C03658=1182.878,246.002,-64.070,-177.311,7.140,148.552
C03659=1182.873,246.251,-64.098,-177.308,7.143,148.552
C03660=1182.869,246.499,-64.123,-177.305,7.145,148.551
C03661=1182.864,246.748,-64.150,-177.303,7.148,148.551
C03662=1182.860,246.996,-64.177,-177.300,7.150,148.551
C03663=1182.856,247.245,-64.204,-177.297,7.153,148.551
C03664=1182.851,247.493,-64.231,-177.295,7.155,148.551
C03665=1182.847,247.742,-64.257,-177.292,7.158,148.551
C03666=1182.842,247.990,-64.284,-177.290,7.160,148.551
C03667=1182.837,248.239,-64.311,-177.287,7.163,148.551
C03668=1182.834,248.487,-64.337,-177.285,7.165,148.550
C03669=1182.829,248.736,-64.364,-177.282,7.168,148.550
C03670=1182.824,248.984,-64.391,-177.279,7.170,148.550
C03671=1182.820,249.233,-64.418,-177.277,7.173,148.550
C03672=1182.815,249.481,-64.444,-177.274,7.175,148.550
C03673=1182.811,249.730,-64.471,-177.271,7.178,148.550
C03674=1182.806,249.978,-64.498,-177.269,7.181,148.550
C03675=1182.803,250.227,-64.525,-177.266,7.182,148.549
C03676=1182.798,250.476,-64.552,-177.263,7.185,148.549
C03677=1182.793,250.724,-64.579,-177.261,7.188,148.549
C03678=1182.789,250.973,-64.606,-177.258,7.190,148.549
C03679=1182.785,251.221,-64.633,-177.256,7.192,148.549
C03680=1182.780,251.469,-64.660,-177.253,7.195,148.549
C03681=1182.775,251.718,-64.687,-177.251,7.197,148.549
C03682=1182.771,251.966,-64.714,-177.248,7.200,148.548
C03683=1182.766,252.215,-64.741,-177.245,7.202,148.548
C03684=1182.763,252.464,-64.768,-177.243,7.205,148.548
C03685=1182.758,252.712,-64.795,-177.240,7.207,148.548
C03686=1182.754,252.961,-64.822,-177.237,7.210,148.548
C03687=1182.749,253.209,-64.850,-177.235,7.213,148.548
C03688=1182.745,253.457,-64.877,-177.232,7.215,148.548
C03689=1182.740,253.706,-64.904,-177.229,7.218,148.547
C03690=1182.737,253.955,-64.931,-177.227,7.220,148.547
C03691=1182.732,254.203,-64.958,-177.224,7.223,148.547
C03692=1182.727,254.452,-64.985,-177.222,7.225,148.547
C03693=1182.723,254.700,-65.012,-177.219,7.228,148.547
C03694=1182.718,254.948,-65.040,-177.216,7.231,148.547
C03695=1182.714,255.196,-65.067,-177.214,7.233,148.547
C03696=1182.710,255.446,-65.094,-177.211,7.236,148.546
C03697=1182.705,255.694,-65.121,-177.209,7.238,148.546
C03698=1182.700,255.943,-65.148,-177.206,7.241,148.546
C03699=1182.697,256.190,-65.176,-177.204,7.243,148.546
C03700=1182.692,256.439,-65.203,-177.201,7.245,148.546
C03701=1182.688,256.688,-65.230,-177.198,7.248,148.546
C03702=1182.684,256.936,-65.258,-177.196,7.251,148.546
C03703=1182.679,257.184,-65.285,-177.193,7.254,148.546
C03704=1182.674,257.433,-65.312,-177.190,7.255,148.545
C03705=1182.670,257.682,-65.339,-177.187,7.258,148.545
C03706=1182.666,257.930,-65.367,-177.185,7.261,148.545
C03707=1182.661,258.178,-65.394,-177.183,7.264,148.545
C03708=1182.657,258.427,-65.421,-177.179,7.266,148.545
C03709=1182.653,258.675,-65.449,-177.177,7.268,148.545
C03710=1182.648,258.924,-65.476,-177.174,7.271,148.545
C03711=1182.644,259.172,-65.504,-177.172,7.273,148.545
C03712=1182.639,259.420,-65.531,-177.170,7.276,148.545
C03713=1182.635,259.669,-65.559,-177.166,7.279,148.544
C03714=1182.631,259.917,-65.586,-177.164,7.281,148.544
C03715=1182.625,260.166,-65.614,-177.161,7.284,148.544
C03716=1182.622,260.415,-65.642,-177.159,7.287,148.544
C03717=1182.617,260.663,-65.669,-177.156,7.289,148.544
C03718=1182.613,260.911,-65.697,-177.153,7.292,148.544
C03719=1182.608,261.160,-65.725,-177.151,7.294,148.544
C03720=1182.604,261.408,-65.752,-177.148,7.297,148.544
C03721=1182.599,261.657,-65.779,-177.146,7.300,148.544
C03722=1182.596,261.905,-65.808,-177.143,7.302,148.543
C03723=1182.590,262.178,-65.838,-177.140,7.305,148.543
C03724=1182.586,262.451,-65.869,-177.138,7.308,148.543
C03725=1182.581,262.724,-65.899,-177.135,7.311,148.543
C03726=1182.577,262.997,-65.929,-177.132,7.314,148.543
C03727=1182.571,263.246,-65.957,-177.129,7.317,148.543
C03728=1182.567,263.493,-65.984,-177.127,7.319,148.543
C03729=1182.563,263.742,-66.012,-177.124,7.322,148.543
C03730=1182.558,263.991,-66.040,-177.121,7.324,148.542
C03731=1182.554,264.238,-66.067,-177.119,7.327,148.542
C03732=1182.550,264.487,-66.096,-177.116,7.329,148.542
C03733=1182.545,264.736,-66.123,-177.113,7.332,148.542
C03734=1182.541,264.984,-66.151,-177.111,7.335,148.542
C03735=1182.537,265.232,-66.179,-177.108,7.338,148.542
C03736=1182.532,265.481,-66.206,-177.106,7.339,148.542
C03737=1182.528,265.730,-66.235,-177.103,7.342,148.542
C03738=1182.523,265.977,-66.263,-177.100,7.345,148.542
C03739=1182.520,266.226,-66.291,-177.098,7.348,148.542
C03740=1182.514,266.475,-66.318,-177.095,7.351,148.542
C03741=1182.510,266.723,-66.346,-177.093,7.354,148.542
C03742=1182.506,266.971,-66.374,-177.090,7.356,148.541
C03743=1182.502,267.219,-66.402,-177.087,7.358,148.541
C03744=1182.497,267.469,-66.430,-177.085,7.361,148.541
C03745=1182.493,267.717,-66.458,-177.082,7.363,148.541
C03746=1182.489,267.965,-66.486,-177.080,7.366,148.541
C03747=1182.484,268.213,-66.514,-177.077,7.369,148.541
C03748=1182.479,268.461,-66.542,-177.075,7.372,148.541
C03749=1182.476,268.710,-66.570,-177.072,7.375,148.541
C03750=1182.471,268.958,-66.599,-177.069,7.378,148.541
C03751=1182.467,269.207,-66.626,-177.067,7.379,148.540
C03752=1182.462,269.455,-66.654,-177.064,7.382,148.540
C03753=1182.458,269.704,-66.683,-177.061,7.385,148.540
C03754=1182.453,269.952,-66.710,-177.059,7.388,148.540
C03755=1182.449,270.201,-66.739,-177.056,7.391,148.540
C03756=1182.445,270.449,-66.767,-177.054,7.394,148.540
C03757=1182.441,270.697,-66.795,-177.051,7.396,148.540
C03758=1182.436,270.945,-66.823,-177.049,7.399,148.540
C03759=1182.432,271.194,-66.852,-177.045,7.401,148.540
C03760=1182.427,271.442,-66.880,-177.043,7.403,148.540
C03761=1182.423,271.691,-66.908,-177.041,7.406,148.540
C03762=1182.418,271.939,-66.937,-177.038,7.409,148.540
C03763=1182.414,272.187,-66.965,-177.036,7.412,148.540
C03764=1182.409,272.436,-66.993,-177.033,7.415,148.540
C03765=1182.405,272.684,-67.021,-177.030,7.418,148.539
C03766=1182.402,272.932,-67.050,-177.028,7.420,148.539
C03767=1182.397,273.180,-67.078,-177.025,7.423,148.539
C03768=1182.393,273.429,-67.107,-177.023,7.426,148.539
C03769=1182.388,273.677,-67.135,-177.020,7.429,148.539
C03770=1182.384,273.926,-67.163,-177.017,7.431,148.539
C03771=1182.379,274.174,-67.191,-177.015,7.433,148.539
C03772=1182.375,274.423,-67.220,-177.012,7.436,148.539
C03773=1182.371,274.671,-67.248,-177.010,7.439,148.539
C03774=1182.366,274.919,-67.277,-177.007,7.442,148.539
C03775=1182.362,275.168,-67.306,-177.004,7.445,148.539
C03776=1182.357,275.416,-67.334,-177.002,7.447,148.539
C03777=1182.354,275.664,-67.362,-176.999,7.450,148.539
C03778=1182.349,275.913,-67.392,-176.997,7.453,148.539
C03779=1182.345,276.160,-67.419,-176.994,7.456,148.539
C03780=1182.341,276.409,-67.448,-176.992,7.458,148.538
C03781=1182.335,276.657,-67.476,-176.989,7.461,148.538
C03782=1182.332,276.905,-67.505,-176.986,7.464,148.538
C03783=1182.328,277.154,-67.534,-176.984,7.466,148.538
C03784=1182.322,277.403,-67.562,-176.981,7.469,148.538
C03785=1182.319,277.650,-67.591,-176.979,7.472,148.538
C03786=1182.315,277.899,-67.620,-176.976,7.475,148.538
C03787=1182.310,278.147,-67.648,-176.974,7.477,148.538
C03788=1182.306,278.395,-67.677,-176.971,7.480,148.538
C03789=1182.302,278.644,-67.706,-176.968,7.483,148.538
C03790=1182.297,278.892,-67.734,-176.965,7.486,148.538
C03791=1182.293,279.141,-67.763,-176.963,7.488,148.538
C03792=1182.288,279.389,-67.792,-176.960,7.491,148.538
C03793=1182.284,279.637,-67.820,-176.957,7.494,148.538
C03794=1182.280,279.886,-67.849,-176.955,7.496,148.538
C03795=1182.276,280.134,-67.879,-176.953,7.499,148.537
C03796=1182.271,280.382,-67.907,-176.950,7.502,148.537
C03797=1182.267,280.630,-67.936,-176.947,7.505,148.537
C03798=1182.263,280.879,-67.965,-176.945,7.507,148.537
C03799=1182.259,281.127,-67.994,-176.942,7.510,148.537
C03800=1182.253,281.375,-68.022,-176.939,7.513,148.537
C03801=1182.250,281.623,-68.051,-176.937,7.516,148.537
C03802=1182.246,281.872,-68.080,-176.935,7.518,148.537
C03803=1182.241,282.120,-68.109,-176.932,7.521,148.537
C03804=1182.236,282.369,-68.138,-176.929,7.524,148.537
C03805=1182.232,282.617,-68.167,-176.926,7.527,148.537
C03806=1182.229,282.865,-68.196,-176.924,7.529,148.537
C03807=1182.224,283.113,-68.224,-176.922,7.532,148.537
C03808=1182.219,283.361,-68.254,-176.919,7.535,148.537
C03809=1182.215,283.610,-68.283,-176.916,7.538,148.537
C03810=1182.211,283.858,-68.312,-176.914,7.541,148.537
C03811=1182.206,284.106,-68.341,-176.911,7.544,148.537
C03812=1182.201,284.355,-68.370,-176.908,7.547,148.537
C03813=1182.198,284.603,-68.399,-176.906,7.550,148.537
C03814=1182.194,284.851,-68.428,-176.904,7.552,148.537
C03815=1182.190,285.099,-68.458,-176.901,7.555,148.537
C03816=1182.185,285.348,-68.486,-176.899,7.558,148.537
C03817=1182.180,285.596,-68.516,-176.896,7.561,148.537
C03818=1182.176,285.844,-68.545,-176.893,7.564,148.537
C03819=1182.172,286.092,-68.574,-176.891,7.566,148.537
C03820=1182.168,286.341,-68.603,-176.888,7.569,148.537
C03821=1182.163,286.589,-68.632,-176.886,7.572,148.537
C03822=1182.159,286.837,-68.662,-176.883,7.575,148.536
C03823=1182.154,287.085,-68.691,-176.881,7.577,148.536
C03824=1182.150,287.334,-68.721,-176.878,7.580,148.536
C03825=1182.146,287.583,-68.749,-176.875,7.583,148.536
C03826=1182.142,287.831,-68.779,-176.872,7.586,148.536
C03827=1182.137,288.105,-68.811,-176.870,7.589,148.536
C03828=1182.132,288.380,-68.844,-176.867,7.592,148.536
C03829=1182.128,288.654,-68.876,-176.864,7.595,148.536
C03830=1182.123,288.929,-68.909,-176.862,7.598,148.536
C03831=1182.118,289.177,-68.938,-176.859,7.601,148.536
C03832=1182.114,289.426,-68.968,-176.856,7.604,148.536
C03833=1182.110,289.673,-68.997,-176.853,7.607,148.536
C03834=1182.105,289.921,-69.026,-176.851,7.610,148.536
C03835=1182.101,290.170,-69.056,-176.849,7.612,148.536
C03836=1182.097,290.418,-69.085,-176.846,7.615,148.536
C03837=1182.093,290.666,-69.115,-176.843,7.618,148.536
C03838=1182.089,290.914,-69.144,-176.841,7.622,148.536
C03839=1182.084,291.163,-69.173,-176.838,7.625,148.536
C03840=1182.080,291.411,-69.203,-176.836,7.627,148.536
C03841=1182.076,291.659,-69.232,-176.833,7.630,148.536
C03842=1182.072,291.908,-69.262,-176.830,7.633,148.536
C03843=1182.067,292.156,-69.292,-176.828,7.636,148.536
C03844=1182.063,292.404,-69.321,-176.825,7.639,148.536
C03845=1182.058,292.652,-69.350,-176.823,7.641,148.536
C03846=1182.054,292.900,-69.380,-176.820,7.644,148.536
C03847=1182.050,293.148,-69.409,-176.817,7.647,148.536
C03848=1182.046,293.396,-69.439,-176.815,7.650,148.536
C03849=1182.042,293.644,-69.469,-176.812,7.653,148.536
C03850=1182.037,293.893,-69.499,-176.810,7.655,148.536
C03851=1182.032,294.141,-69.528,-176.808,7.658,148.536
C03852=1182.028,294.390,-69.558,-176.805,7.661,148.536
C03853=1182.024,294.637,-69.588,-176.802,7.664,148.536
C03854=1182.020,294.885,-69.618,-176.799,7.667,148.536
C03855=1182.015,295.134,-69.648,-176.797,7.670,148.536
C03856=1182.011,295.382,-69.677,-176.795,7.673,148.536
C03857=1182.007,295.630,-69.707,-176.792,7.676,148.536
C03858=1182.003,295.878,-69.737,-176.790,7.679,148.536
C03859=1181.998,296.127,-69.767,-176.787,7.682,148.536
C03860=1181.994,296.375,-69.796,-176.784,7.685,148.536
C03861=1181.990,296.623,-69.826,-176.781,7.688,148.536
C03862=1181.986,296.871,-69.856,-176.779,7.690,148.536
C03863=1181.981,297.120,-69.886,-176.777,7.693,148.536
C03864=1181.978,297.368,-69.916,-176.774,7.696,148.536
C03865=1181.974,297.616,-69.946,-176.771,7.699,148.536
C03866=1181.969,297.864,-69.977,-176.769,7.702,148.536
C03867=1181.965,298.112,-70.006,-176.766,7.705,148.536
C03868=1181.961,298.361,-70.035,-176.764,7.707,148.536
C03869=1181.956,298.609,-70.066,-176.762,7.711,148.536
C03870=1181.952,298.857,-70.096,-176.759,7.714,148.536
C03871=1181.948,299.105,-70.126,-176.756,7.717,148.536
C03872=1181.943,299.353,-70.156,-176.753,7.720,148.536
C03873=1181.939,299.601,-70.186,-176.751,7.723,148.536
C03874=1181.935,299.849,-70.216,-176.749,7.725,148.536
C03875=1181.930,300.097,-70.246,-176.746,7.728,148.536
C03876=1181.926,300.345,-70.276,-176.744,7.731,148.536
C03877=1181.922,300.594,-70.307,-176.741,7.734,148.536
C03878=1181.918,300.842,-70.336,-176.738,7.737,148.536
C03879=1181.913,301.090,-70.367,-176.735,7.740,148.536
C03880=1181.909,301.338,-70.397,-176.734,7.743,148.536
C03881=1181.905,301.586,-70.427,-176.731,7.746,148.536
C03882=1181.900,301.835,-70.457,-176.728,7.749,148.536
C03883=1181.896,302.082,-70.487,-176.726,7.752,148.536
C03884=1181.892,302.330,-70.518,-176.723,7.755,148.536
C03885=1181.888,302.579,-70.548,-176.721,7.758,148.536
C03886=1181.884,302.827,-70.578,-176.718,7.761,148.536
C03887=1181.880,303.075,-70.608,-176.716,7.763,148.536
C03888=1181.875,303.323,-70.638,-176.713,7.766,148.536
C03889=1181.871,303.571,-70.669,-176.710,7.769,148.536
C03890=1181.866,303.819,-70.699,-176.708,7.772,148.536
C03891=1181.863,304.068,-70.729,-176.705,7.775,148.536
C03892=1181.858,304.316,-70.760,-176.703,7.778,148.536
C03893=1181.854,304.564,-70.790,-176.700,7.781,148.536
C03894=1181.849,304.812,-70.820,-176.698,7.785,148.536
C03895=1181.845,305.060,-70.851,-176.695,7.787,148.536
C03896=1181.841,305.308,-70.881,-176.693,7.790,148.536
C03897=1181.837,305.556,-70.912,-176.690,7.793,148.536
C03898=1181.833,305.804,-70.942,-176.688,7.796,148.536
C03899=1181.828,306.053,-70.972,-176.685,7.799,148.536
C03900=1181.823,306.301,-71.003,-176.682,7.802,148.536
C03901=1181.820,306.549,-71.034,-176.680,7.805,148.536
C03902=1181.816,306.797,-71.065,-176.677,7.808,148.537
C03903=1181.812,307.045,-71.095,-176.675,7.811,148.536
C03904=1181.807,307.292,-71.125,-176.672,7.814,148.536
C03905=1181.802,307.540,-71.156,-176.670,7.817,148.536
C03906=1181.799,307.789,-71.186,-176.667,7.820,148.537
C03907=1181.794,308.037,-71.217,-176.665,7.823,148.537
C03908=1181.790,308.285,-71.248,-176.662,7.826,148.537
C03909=1181.786,308.533,-71.278,-176.660,7.829,148.537
C03910=1181.782,308.782,-71.309,-176.657,7.832,148.537
C03911=1181.777,309.030,-71.340,-176.655,7.834,148.537
C03912=1181.773,309.277,-71.370,-176.652,7.837,148.537
C03913=1181.769,309.526,-71.401,-176.650,7.841,148.537
C03914=1181.765,309.774,-71.432,-176.647,7.844,148.537
C03915=1181.760,310.022,-71.462,-176.644,7.847,148.537
C03916=1181.757,310.270,-71.493,-176.642,7.850,148.537
C03917=1181.752,310.518,-71.524,-176.639,7.853,148.537
C03918=1181.748,310.766,-71.555,-176.637,7.856,148.537
C03919=1181.743,311.014,-71.585,-176.635,7.859,148.537
C03920=1181.740,311.262,-71.616,-176.632,7.861,148.537
C03921=1181.735,311.510,-71.647,-176.630,7.864,148.537
C03922=1181.731,311.758,-71.678,-176.627,7.868,148.537
C03923=1181.727,312.006,-71.709,-176.625,7.871,148.537
C03924=1181.722,312.254,-71.740,-176.622,7.874,148.537
C03925=1181.718,312.502,-71.770,-176.620,7.877,148.537
C03926=1181.714,312.751,-71.801,-176.617,7.880,148.537
C03927=1181.710,312.999,-71.832,-176.614,7.883,148.537
C03928=1181.706,313.247,-71.864,-176.612,7.886,148.538
C03929=1181.701,313.495,-71.895,-176.609,7.889,148.538
C03930=1181.697,313.743,-71.925,-176.607,7.892,148.538
C03931=1181.693,314.019,-71.960,-176.604,7.896,148.538
C03932=1181.688,314.296,-71.994,-176.602,7.899,148.538
C03933=1181.683,314.573,-72.029,-176.598,7.902,148.538
C03934=1181.678,314.849,-72.064,-176.596,7.905,148.538
C03935=1181.674,315.097,-72.095,-176.593,7.909,148.538
C03936=1181.670,315.345,-72.125,-176.591,7.912,148.538
C03937=1181.666,315.593,-72.157,-176.588,7.915,148.538
C03938=1181.661,315.841,-72.188,-176.586,7.918,148.538
C03939=1181.657,316.090,-72.219,-176.583,7.921,148.538
C03940=1181.653,316.337,-72.251,-176.581,7.924,148.538
C03941=1181.648,316.585,-72.281,-176.578,7.927,148.538
C03942=1181.644,316.834,-72.313,-176.576,7.930,148.538
C03943=1181.640,317.081,-72.344,-176.573,7.933,148.539
C03944=1181.637,317.330,-72.375,-176.571,7.936,148.539
C03945=1181.633,317.577,-72.406,-176.569,7.939,148.539
C03946=1181.629,317.826,-72.437,-176.566,7.942,148.539
C03947=1181.624,318.073,-72.469,-176.563,7.945,148.539
C03948=1181.620,318.322,-72.500,-176.561,7.948,148.539
C03949=1181.616,318.569,-72.531,-176.558,7.951,148.539
C03950=1181.612,318.818,-72.562,-176.556,7.955,148.539
C03951=1181.607,319.066,-72.593,-176.553,7.958,148.539
C03952=1181.604,319.314,-72.625,-176.551,7.961,148.539
C03953=1181.599,319.561,-72.657,-176.549,7.963,148.539
C03954=1181.595,319.810,-72.688,-176.546,7.966,148.539
C03955=1181.590,320.057,-72.720,-176.544,7.970,148.539
C03956=1181.586,320.306,-72.751,-176.541,7.973,148.539
C03957=1181.582,320.553,-72.782,-176.539,7.976,148.540
C03958=1181.578,320.802,-72.813,-176.536,7.979,148.540
C03959=1181.574,321.049,-72.845,-176.534,7.982,148.540
C03960=1181.570,321.297,-72.877,-176.531,7.985,148.540
C03961=1181.565,321.545,-72.907,-176.529,7.989,148.540
C03962=1181.562,321.793,-72.939,-176.526,7.992,148.540
C03963=1181.557,322.041,-72.971,-176.523,7.995,148.540
C03964=1181.552,322.290,-73.003,-176.521,7.998,148.540
C03965=1181.548,322.537,-73.034,-176.518,8.001,148.540
C03966=1181.544,322.785,-73.066,-176.516,8.004,148.540
C03967=1181.540,323.034,-73.097,-176.513,8.007,148.540
C03968=1181.536,323.281,-73.128,-176.511,8.010,148.541
C03969=1181.532,323.529,-73.160,-176.508,8.013,148.541
C03970=1181.528,323.776,-73.192,-176.507,8.016,148.541
C03971=1181.523,324.025,-73.224,-176.504,8.019,148.541
C03972=1181.520,324.273,-73.255,-176.502,8.022,148.541
C03973=1181.515,324.521,-73.287,-176.499,8.025,148.541
C03974=1181.512,324.769,-73.319,-176.497,8.029,148.541
C03975=1181.507,325.017,-73.349,-176.494,8.032,148.541
C03976=1181.503,325.265,-73.382,-176.492,8.035,148.541
C03977=1181.499,325.513,-73.414,-176.490,8.038,148.542
C03978=1181.495,325.760,-73.445,-176.487,8.041,148.542
C03979=1181.491,326.008,-73.477,-176.485,8.044,148.542
C03980=1181.486,326.256,-73.509,-176.482,8.047,148.542
C03981=1181.482,326.504,-73.541,-176.480,8.051,148.542
C03982=1181.478,326.752,-73.573,-176.477,8.054,148.542
C03983=1181.473,327.000,-73.604,-176.475,8.057,148.542
C03984=1181.469,327.249,-73.636,-176.472,8.060,148.542
C03985=1181.466,327.497,-73.668,-176.470,8.063,148.542
C03986=1181.461,327.744,-73.700,-176.467,8.066,148.542
C03987=1181.457,327.992,-73.732,-176.465,8.070,148.543
C03988=1181.453,328.240,-73.764,-176.462,8.073,148.543
C03989=1181.448,328.488,-73.796,-176.460,8.076,148.543
C03990=1181.444,328.736,-73.828,-176.457,8.079,148.543
C03991=1181.441,328.984,-73.859,-176.455,8.082,148.543
C03992=1181.436,329.232,-73.891,-176.452,8.086,148.543
C03993=1181.432,329.480,-73.923,-176.450,8.089,148.543
C03994=1181.428,329.728,-73.955,-176.447,8.092,148.543
C03995=1181.424,329.975,-73.988,-176.445,8.095,148.544
C03996=1181.420,330.223,-74.020,-176.443,8.097,148.544
C03997=1181.415,330.471,-74.052,-176.441,8.101,148.544
C03998=1181.412,330.719,-74.084,-176.439,8.104,148.544
C03999=1181.407,330.967,-74.116,-176.436,8.107,148.544
C04000=1181.403,331.215,-74.148,-176.434,8.110,148.544
C04001=1181.399,331.463,-74.180,-176.431,8.114,148.544
C04002=1181.395,331.711,-74.212,-176.429,8.117,148.544
C04003=1181.391,331.958,-74.244,-176.426,8.120,148.545
C04004=1181.386,332.206,-74.277,-176.424,8.123,148.545
C04005=1181.383,332.454,-74.309,-176.421,8.126,148.545
C04006=1181.378,332.703,-74.341,-176.419,8.130,148.545
C04007=1181.374,332.950,-74.373,-176.417,8.133,148.545
C04008=1181.370,333.198,-74.406,-176.414,8.136,148.545
C04009=1181.366,333.446,-74.438,-176.412,8.139,148.545
C04010=1181.362,333.694,-74.470,-176.410,8.143,148.546
C04011=1181.358,333.941,-74.502,-176.407,8.146,148.546
C04012=1181.353,334.189,-74.535,-176.405,8.149,148.546
C04013=1181.349,334.437,-74.567,-176.402,8.152,148.546
C04014=1181.345,334.686,-74.599,-176.400,8.155,148.546
C04015=1181.342,334.933,-74.632,-176.397,8.159,148.546
C04016=1181.337,335.181,-74.664,-176.395,8.162,148.546
C04017=1181.332,335.428,-74.697,-176.393,8.165,148.547
C04018=1181.329,335.676,-74.729,-176.390,8.168,148.547
C04019=1181.324,335.925,-74.761,-176.388,8.171,148.547
C04020=1181.321,336.172,-74.794,-176.386,8.175,148.547
C04021=1181.316,336.421,-74.826,-176.383,8.178,148.547
C04022=1181.312,336.668,-74.859,-176.381,8.181,148.547
C04023=1181.308,336.916,-74.891,-176.378,8.184,148.548
C04024=1181.304,337.164,-74.923,-176.376,8.188,148.548
C04025=1181.299,337.412,-74.956,-176.374,8.191,148.548
C04026=1181.296,337.660,-74.988,-176.371,8.194,148.548
C04027=1181.292,337.908,-75.021,-176.369,8.197,148.548
C04028=1181.288,338.156,-75.053,-176.367,8.201,148.548
C04029=1181.283,338.403,-75.086,-176.364,8.204,148.549
C04030=1181.279,338.650,-75.119,-176.362,8.207,148.549
C04031=1181.275,338.899,-75.152,-176.359,8.210,148.549
C04032=1181.271,339.146,-75.184,-176.357,8.214,148.549
C04033=1181.267,339.394,-75.217,-176.355,8.217,148.549
C04034=1181.263,339.642,-75.250,-176.353,8.220,148.549
C04035=1181.258,339.921,-75.286,-176.350,8.224,148.550
C04036=1181.254,340.201,-75.323,-176.347,8.227,148.550
C04037=1181.249,340.479,-75.360,-176.344,8.232,148.550
C04038=1181.244,340.758,-75.396,-176.342,8.235,148.550
C04039=1181.240,341.006,-75.429,-176.340,8.238,148.550
C04040=1181.236,341.253,-75.463,-176.337,8.241,148.551
C04041=1181.232,341.502,-75.495,-176.335,8.245,148.551
C04042=1181.227,341.750,-75.528,-176.333,8.248,148.551
C04043=1181.224,341.997,-75.561,-176.330,8.251,148.551
C04044=1181.220,342.245,-75.593,-176.328,8.254,148.551
C04045=1181.215,342.493,-75.626,-176.326,8.258,148.552
C04046=1181.211,342.741,-75.660,-176.323,8.261,148.552
C04047=1181.207,342.989,-75.693,-176.321,8.264,148.552
C04048=1181.202,343.236,-75.725,-176.319,8.268,148.552
C04049=1181.199,343.484,-75.757,-176.317,8.271,148.552
C04050=1181.195,343.731,-75.790,-176.314,8.274,148.553
C04051=1181.190,343.979,-75.824,-176.312,8.278,148.553
C04052=1181.186,344.227,-75.857,-176.310,8.281,148.553
C04053=1181.182,344.475,-75.889,-176.307,8.285,148.553
C04054=1181.178,344.723,-75.922,-176.305,8.288,148.554
C04055=1181.174,344.971,-75.956,-176.302,8.292,148.554
C04056=1181.169,345.218,-75.989,-176.300,8.295,148.554
C04057=1181.165,345.466,-76.022,-176.298,8.298,148.554
C04058=1181.162,345.713,-76.054,-176.296,8.302,148.554
C04059=1181.158,345.961,-76.088,-176.293,8.305,148.555
C04060=1181.154,346.209,-76.121,-176.291,8.308,148.555
C04061=1181.149,346.457,-76.154,-176.289,8.312,148.555
C04062=1181.145,346.704,-76.187,-176.287,8.315,148.555
C04063=1181.142,346.953,-76.221,-176.284,8.318,148.555
C04064=1181.138,347.201,-76.254,-176.282,8.322,148.556
C04065=1181.134,347.448,-76.287,-176.280,8.325,148.556
C04066=1181.129,347.696,-76.320,-176.278,8.328,148.556
C04067=1181.125,347.944,-76.353,-176.275,8.331,148.556
C04068=1181.121,348.191,-76.386,-176.273,8.335,148.557
C04069=1181.117,348.439,-76.419,-176.271,8.338,148.557
C04070=1181.113,348.687,-76.453,-176.269,8.341,148.557
C04071=1181.109,348.935,-76.486,-176.266,8.345,148.557
C04072=1181.105,349.182,-76.519,-176.264,8.348,148.557
C04073=1181.100,349.430,-76.552,-176.262,8.351,148.558
C04074=1181.096,349.678,-76.585,-176.259,8.355,148.558
C04075=1181.092,349.926,-76.618,-176.258,8.358,148.558
C04076=1181.087,350.174,-76.652,-176.255,8.362,148.559
C04077=1181.084,350.421,-76.686,-176.253,8.365,148.559
C04078=1181.080,350.669,-76.720,-176.250,8.369,148.559
C04079=1181.076,350.917,-76.753,-176.248,8.372,148.559
C04080=1181.072,351.165,-76.786,-176.246,8.376,148.559
C04081=1181.068,351.412,-76.819,-176.244,8.379,148.560
C04082=1181.064,351.659,-76.853,-176.242,8.383,148.560
C04083=1181.060,351.907,-76.886,-176.239,8.386,148.560
C04084=1181.056,352.156,-76.920,-176.237,8.389,148.561
C04085=1181.051,352.404,-76.953,-176.235,8.393,148.561
C04086=1181.047,352.651,-76.987,-176.233,8.396,148.561
C04087=1181.043,352.898,-77.020,-176.231,8.399,148.561
C04088=1181.039,353.146,-77.053,-176.229,8.403,148.562
C04089=1181.035,353.393,-77.087,-176.226,8.406,148.562
C04090=1181.031,353.641,-77.121,-176.224,8.409,148.562
C04091=1181.027,353.890,-77.155,-176.222,8.413,148.562
C04092=1181.023,354.137,-77.189,-176.220,8.416,148.563
C04093=1181.019,354.385,-77.222,-176.218,8.420,148.563
C04094=1181.015,354.632,-77.255,-176.216,8.423,148.563
C04095=1181.011,354.879,-77.289,-176.213,8.427,148.564
C04096=1181.007,355.128,-77.323,-176.211,8.431,148.564
C04097=1181.003,355.375,-77.357,-176.209,8.434,148.564
C04098=1180.999,355.623,-77.390,-176.207,8.438,148.564
C04099=1180.994,355.871,-77.423,-176.204,8.441,148.565
C04100=1180.990,356.119,-77.458,-176.202,8.444,148.565
C04101=1180.986,356.367,-77.491,-176.200,8.448,148.565
C04102=1180.983,356.614,-77.525,-176.198,8.451,148.566
C04103=1180.978,356.861,-77.558,-176.196,8.455,148.566
C04104=1180.974,357.109,-77.592,-176.194,8.458,148.566
C04105=1180.970,357.357,-77.626,-176.192,8.461,148.566
C04106=1180.966,357.604,-77.660,-176.190,8.465,148.567
C04107=1180.962,357.852,-77.694,-176.188,8.468,148.567
C04108=1180.958,358.100,-77.728,-176.186,8.472,148.568
C04109=1180.954,358.347,-77.762,-176.183,8.476,148.568
C04110=1180.950,358.595,-77.795,-176.181,8.479,148.568
C04111=1180.946,358.843,-77.829,-176.179,8.483,148.568
C04112=1180.942,359.091,-77.863,-176.177,8.486,148.569
C04113=1180.938,359.338,-77.897,-176.175,8.490,148.569
C04114=1180.934,359.585,-77.931,-176.173,8.493,148.569
C04115=1180.930,359.834,-77.965,-176.171,8.497,148.570
C04116=1180.926,360.081,-77.999,-176.169,8.500,148.570
C04117=1180.922,360.328,-78.033,-176.167,8.504,148.570
C04118=1180.917,360.576,-78.067,-176.165,8.507,148.571
C04119=1180.914,360.824,-78.101,-176.163,8.511,148.571
C04120=1180.910,361.071,-78.135,-176.161,8.514,148.572
C04121=1180.905,361.319,-78.169,-176.159,8.518,148.572
C04122=1180.902,361.567,-78.203,-176.157,8.521,148.572
C04123=1180.897,361.815,-78.237,-176.155,8.525,148.573
C04124=1180.893,362.062,-78.271,-176.153,8.528,148.573
C04125=1180.889,362.310,-78.306,-176.151,8.532,148.573
C04126=1180.885,362.558,-78.339,-176.149,8.536,148.574
C04127=1180.881,362.806,-78.374,-176.147,8.539,148.574
C04128=1180.878,363.053,-78.408,-176.145,8.542,148.574
C04129=1180.874,363.300,-78.442,-176.143,8.546,148.575
C04130=1180.870,363.548,-78.477,-176.141,8.550,148.575
C04131=1180.866,363.796,-78.510,-176.139,8.553,148.576
C04132=1180.861,364.043,-78.544,-176.137,8.557,148.576
C04133=1180.858,364.291,-78.579,-176.135,8.560,148.576
C04134=1180.853,364.538,-78.613,-176.134,8.564,148.577
C04135=1180.849,364.787,-78.648,-176.132,8.567,148.577
C04136=1180.845,365.034,-78.682,-176.130,8.571,148.578
C04137=1180.841,365.281,-78.716,-176.128,8.575,148.578
C04138=1180.838,365.529,-78.750,-176.126,8.578,148.578
C04139=1180.833,365.811,-78.790,-176.124,8.582,148.579
C04140=1180.828,366.093,-78.828,-176.123,8.586,148.579
C04141=1180.823,366.374,-78.867,-176.120,8.590,148.580
C04142=1180.819,366.655,-78.906,-176.118,8.594,148.580
C04143=1180.815,366.903,-78.941,-176.117,8.597,148.581
C04144=1180.811,367.151,-78.975,-176.115,8.601,148.581
C04145=1180.807,367.398,-79.009,-176.113,8.604,148.582
C04146=1180.803,367.646,-79.044,-176.111,8.608,148.582
C04147=1180.799,367.893,-79.078,-176.109,8.612,148.582
C04148=1180.795,368.141,-79.113,-176.108,8.615,148.583
C04149=1180.791,368.389,-79.147,-176.107,8.618,148.583
C04150=1180.787,368.635,-79.182,-176.105,8.622,148.584
C04151=1180.783,368.883,-79.217,-176.103,8.626,148.584
C04152=1180.779,369.131,-79.251,-176.101,8.629,148.585
C04153=1180.775,369.379,-79.286,-176.099,8.633,148.585
C04154=1180.771,369.626,-79.320,-176.098,8.636,148.586
C04155=1180.767,369.874,-79.355,-176.097,8.640,148.586
C04156=1180.763,370.121,-79.389,-176.095,8.643,148.587
C04157=1180.759,370.369,-79.424,-176.093,8.647,148.587
C04158=1180.755,370.616,-79.459,-176.092,8.650,148.587
C04159=1180.751,370.864,-79.493,-176.090,8.654,148.588
C04160=1180.747,371.112,-79.527,-176.089,8.657,148.588
C04161=1180.743,371.360,-79.562,-176.087,8.661,148.589
C04162=1180.738,371.607,-79.597,-176.086,8.664,148.589
C04163=1180.735,371.854,-79.632,-176.084,8.668,148.590
C04164=1180.731,372.102,-79.666,-176.083,8.671,148.591
C04165=1180.727,372.350,-79.701,-176.082,8.674,148.591
C04166=1180.722,372.597,-79.735,-176.080,8.678,148.591
C04167=1180.719,372.844,-79.770,-176.078,8.682,148.592
C04168=1180.715,373.092,-79.805,-176.077,8.685,148.592
C04169=1180.711,373.340,-79.840,-176.076,8.688,148.593
C04170=1180.707,373.587,-79.875,-176.074,8.692,148.593
C04171=1180.703,373.835,-79.909,-176.073,8.695,148.594
C04172=1180.699,374.083,-79.944,-176.071,8.699,148.594
C04173=1180.695,374.329,-79.979,-176.070,8.703,148.595
C04174=1180.691,374.578,-80.014,-176.069,8.706,148.596
C04175=1180.687,374.825,-80.048,-176.067,8.709,148.596
C04176=1180.683,375.073,-80.084,-176.066,8.713,148.597
C04177=1180.679,375.320,-80.118,-176.065,8.716,148.597
C04178=1180.675,375.568,-80.153,-176.064,8.719,148.598
C04179=1180.671,375.815,-80.188,-176.062,8.723,148.598
C04180=1180.667,376.063,-80.223,-176.061,8.726,148.599
C04181=1180.663,376.310,-80.258,-176.060,8.730,148.599
C04182=1180.659,376.558,-80.293,-176.059,8.733,148.600
C04183=1180.656,376.805,-80.328,-176.058,8.737,148.601
C04184=1180.652,377.053,-80.363,-176.056,8.740,148.601
C04185=1180.647,377.300,-80.397,-176.055,8.744,148.602
C04186=1180.644,377.548,-80.433,-176.054,8.747,148.602
C04187=1180.639,377.795,-80.467,-176.053,8.751,148.603
C04188=1180.635,378.043,-80.503,-176.052,8.754,148.603
C04189=1180.631,378.291,-80.537,-176.051,8.757,148.604
C04190=1180.627,378.538,-80.573,-176.049,8.760,148.604
C04191=1180.623,378.786,-80.607,-176.048,8.764,148.605
C04192=1180.619,379.033,-80.643,-176.048,8.767,148.606
C04193=1180.615,379.281,-80.677,-176.046,8.771,148.606
C04194=1180.611,379.528,-80.713,-176.045,8.774,148.607
C04195=1180.608,379.775,-80.748,-176.045,8.777,148.607
C04196=1180.604,380.023,-80.782,-176.043,8.781,148.608
C04197=1180.599,380.270,-80.818,-176.042,8.784,148.609
C04198=1180.595,380.518,-80.852,-176.042,8.787,148.609
C04199=1180.592,380.765,-80.888,-176.041,8.790,148.610
C04200=1180.588,381.012,-80.923,-176.039,8.794,148.610
C04201=1180.584,381.260,-80.958,-176.038,8.797,148.611
C04202=1180.580,381.508,-80.994,-176.038,8.800,148.612
C04203=1180.575,381.755,-81.028,-176.037,8.803,148.612
C04204=1180.572,382.003,-81.064,-176.036,8.806,148.613
C04205=1180.568,382.250,-81.099,-176.035,8.809,148.613
C04206=1180.563,382.497,-81.134,-176.034,8.812,148.614
C04207=1180.560,382.745,-81.169,-176.033,8.816,148.614
C04208=1180.556,382.992,-81.205,-176.032,8.819,148.615
C04209=1180.552,383.240,-81.239,-176.032,8.823,148.616
C04210=1180.548,383.487,-81.275,-176.031,8.826,148.616
C04211=1180.544,383.735,-81.310,-176.030,8.829,148.617
C04212=1180.540,383.982,-81.345,-176.029,8.832,148.618
C04213=1180.536,384.230,-81.380,-176.028,8.835,148.618
C04214=1180.532,384.477,-81.416,-176.028,8.838,148.619
C04215=1180.528,384.724,-81.451,-176.027,8.842,148.620
C04216=1180.523,384.973,-81.486,-176.026,8.845,148.620
C04217=1180.520,385.220,-81.522,-176.026,8.848,148.621
C04218=1180.516,385.468,-81.557,-176.025,8.851,148.621
C04219=1180.512,385.714,-81.593,-176.025,8.854,148.622
C04220=1180.508,385.962,-81.627,-176.024,8.857,148.623
C04221=1180.504,386.210,-81.663,-176.023,8.860,148.623
C04222=1180.500,386.457,-81.698,-176.023,8.863,148.624
C04223=1180.496,386.704,-81.734,-176.022,8.866,148.625
C04224=1180.492,386.952,-81.769,-176.021,8.869,148.625
C04225=1180.489,387.200,-81.804,-176.021,8.872,148.626
C04226=1180.484,387.447,-81.839,-176.021,8.875,148.626
C04227=1180.481,387.694,-81.875,-176.020,8.878,148.627
C04228=1180.476,387.942,-81.911,-176.020,8.881,148.628
C04229=1180.472,388.189,-81.946,-176.019,8.884,148.628
C04230=1180.468,388.437,-81.981,-176.019,8.887,148.629
C04231=1180.464,388.684,-82.017,-176.018,8.890,148.630
C04232=1180.461,388.932,-82.052,-176.018,8.893,148.630
C04233=1180.456,389.179,-82.087,-176.017,8.896,148.631
C04234=1180.453,389.426,-82.123,-176.018,8.898,148.632
C04235=1180.449,389.674,-82.158,-176.017,8.902,148.632
C04236=1180.445,389.922,-82.195,-176.016,8.905,148.633
C04237=1180.440,390.169,-82.229,-176.016,8.907,148.634
C04238=1180.436,390.416,-82.265,-176.016,8.911,148.634
C04239=1180.433,390.664,-82.300,-176.015,8.913,148.635
C04240=1180.429,390.911,-82.336,-176.015,8.916,148.636
C04241=1180.425,391.158,-82.371,-176.015,8.918,148.636
C04242=1180.421,391.406,-82.406,-176.014,8.922,148.637
C04243=1180.416,391.691,-82.447,-176.015,8.924,148.638
C04244=1180.412,391.974,-82.488,-176.014,8.928,148.638
C04245=1180.408,392.259,-82.529,-176.013,8.931,148.639
C04246=1180.403,392.543,-82.570,-176.013,8.934,148.640
C04247=1180.399,392.790,-82.606,-176.013,8.937,148.641
C04248=1180.395,393.038,-82.641,-176.013,8.939,148.641
C04249=1180.392,393.285,-82.677,-176.012,8.943,148.642
C04250=1180.387,393.532,-82.712,-176.012,8.945,148.642
C04251=1180.383,393.780,-82.748,-176.012,8.947,148.643
C04252=1180.379,394.027,-82.784,-176.012,8.951,148.644
C04253=1180.376,394.275,-82.819,-176.012,8.953,148.644
C04254=1180.371,394.521,-82.854,-176.012,8.956,148.645
C04255=1180.368,394.769,-82.890,-176.011,8.959,148.646
C04256=1180.363,395.017,-82.926,-176.011,8.961,148.646
C04257=1180.360,395.264,-82.961,-176.011,8.964,148.647
C04258=1180.356,395.512,-82.997,-176.011,8.966,148.648
C04259=1180.352,395.759,-83.032,-176.011,8.969,148.648
C04260=1180.347,396.006,-83.068,-176.010,8.972,148.649
C04261=1180.344,396.254,-83.104,-176.011,8.974,148.650
C04262=1180.340,396.501,-83.139,-176.010,8.977,148.650
C04263=1180.336,396.749,-83.175,-176.011,8.979,148.651
C04264=1180.331,396.996,-83.211,-176.010,8.981,148.651
C04265=1180.328,397.244,-83.246,-176.010,8.984,148.652
C04266=1180.324,397.491,-83.282,-176.011,8.987,148.653
C04267=1180.320,397.739,-83.317,-176.010,8.989,148.653
C04268=1180.316,397.986,-83.354,-176.010,8.992,148.654
C04269=1180.312,398.233,-83.389,-176.010,8.995,148.655
C04270=1180.308,398.481,-83.424,-176.010,8.997,148.655
C04271=1180.304,398.728,-83.460,-176.010,8.999,148.656
C04272=1180.300,398.976,-83.496,-176.010,9.002,148.657
C04273=1180.296,399.223,-83.532,-176.010,9.004,148.657
C04274=1180.293,399.470,-83.568,-176.010,9.007,148.658
C04275=1180.289,399.717,-83.603,-176.010,9.009,148.659
C04276=1180.284,399.965,-83.639,-176.010,9.012,148.659
C04277=1180.281,400.212,-83.675,-176.010,9.014,148.660
C04278=1180.277,400.460,-83.710,-176.010,9.016,148.660
C04279=1180.273,400.708,-83.746,-176.010,9.019,148.661
C04280=1180.268,400.955,-83.782,-176.010,9.020,148.662
C04281=1180.265,401.202,-83.817,-176.010,9.023,148.662
C04282=1180.261,401.450,-83.853,-176.010,9.026,148.663
C04283=1180.257,401.697,-83.889,-176.010,9.028,148.663
C04284=1180.253,401.944,-83.925,-176.010,9.030,148.664
C04285=1180.250,402.192,-83.961,-176.010,9.033,148.665
C04286=1180.245,402.440,-83.997,-176.010,9.035,148.665
C04287=1180.241,402.686,-84.032,-176.010,9.037,148.666
C04288=1180.237,402.934,-84.067,-176.010,9.040,148.667
C04289=1180.233,403.182,-84.104,-176.010,9.041,148.667
C04290=1180.229,403.429,-84.139,-176.011,9.044,148.668
C04291=1180.226,403.676,-84.175,-176.010,9.046,148.668
C04292=1180.221,403.924,-84.212,-176.010,9.049,148.669
C04293=1180.217,404.171,-84.247,-176.010,9.051,148.670
C04294=1180.214,404.418,-84.282,-176.011,9.053,148.670
C04295=1180.210,404.666,-84.318,-176.011,9.055,148.671
C04296=1180.205,404.913,-84.354,-176.011,9.058,148.672
C04297=1180.202,405.160,-84.390,-176.011,9.060,148.672
C04298=1180.198,405.408,-84.426,-176.011,9.061,148.672
C04299=1180.194,405.656,-84.462,-176.011,9.064,148.673
C04300=1180.190,405.902,-84.497,-176.011,9.066,148.674
C04301=1180.186,406.150,-84.533,-176.011,9.069,148.674
C04302=1180.182,406.397,-84.570,-176.011,9.070,148.675
C04303=1180.178,406.645,-84.605,-176.011,9.073,148.676
C04304=1180.174,406.892,-84.641,-176.011,9.075,148.676
C04305=1180.170,407.140,-84.677,-176.012,9.077,148.677
C04306=1180.167,407.387,-84.712,-176.012,9.079,148.677
C04307=1180.163,407.635,-84.749,-176.011,9.081,148.678
C04308=1180.158,407.881,-84.784,-176.012,9.083,148.679
C04309=1180.155,408.129,-84.820,-176.012,9.085,148.679
C04310=1180.150,408.377,-84.856,-176.011,9.088,148.680
C04311=1180.147,408.624,-84.892,-176.012,9.089,148.680
C04312=1180.143,408.871,-84.928,-176.012,9.092,148.681
C04313=1180.139,409.119,-84.964,-176.012,9.094,148.681
C04314=1180.135,409.366,-85.000,-176.012,9.096,148.682
C04315=1180.132,409.613,-85.036,-176.012,9.098,148.682
C04316=1180.127,409.860,-85.072,-176.012,9.100,148.683
C04317=1180.123,410.108,-85.107,-176.013,9.102,148.684
C04318=1180.119,410.356,-85.143,-176.012,9.104,148.684
C04319=1180.115,410.603,-85.180,-176.013,9.106,148.685
C04320=1180.112,410.850,-85.215,-176.013,9.108,148.685
C04321=1180.107,411.098,-85.251,-176.013,9.110,148.686
C04322=1180.104,411.345,-85.287,-176.013,9.112,148.686
C04323=1180.100,411.592,-85.323,-176.013,9.114,148.687
C04324=1180.096,411.840,-85.359,-176.013,9.116,148.687
C04325=1180.092,412.087,-85.394,-176.013,9.118,148.688
C04326=1180.087,412.334,-85.431,-176.014,9.120,148.689
C04327=1180.084,412.582,-85.467,-176.013,9.122,148.689
C04328=1180.080,412.829,-85.502,-176.014,9.124,148.690
C04329=1180.076,413.077,-85.538,-176.013,9.126,148.690
C04330=1180.072,413.324,-85.575,-176.014,9.128,148.691
C04331=1180.068,413.572,-85.611,-176.014,9.130,148.691
C04332=1180.064,413.819,-85.646,-176.014,9.131,148.692
C04333=1180.061,414.066,-85.683,-176.014,9.134,148.692
C04334=1180.057,414.314,-85.719,-176.014,9.135,148.693
C04335=1180.052,414.561,-85.754,-176.014,9.138,148.693
C04336=1180.048,414.808,-85.791,-176.015,9.139,148.694
C04337=1180.045,415.055,-85.826,-176.014,9.141,148.694
C04338=1180.040,415.303,-85.863,-176.015,9.143,148.695
C04339=1180.037,415.533,-85.896,-176.014,9.145,148.695
C04340=1180.033,415.763,-85.929,-176.015,9.146,148.696
C04341=1180.032,415.993,-85.963,-176.015,9.149,148.696
C04342=1180.030,416.224,-85.996,-176.015,9.150,148.697
C04343=1180.029,416.454,-86.030,-176.015,9.151,148.697
C04344=1180.030,416.684,-86.062,-176.015,9.153,148.698
C04345=1180.031,416.913,-86.095,-176.015,9.155,148.698
C04346=1180.034,417.142,-86.128,-176.015,9.156,148.699
C04347=1179.612,417.144,-86.171,-176.018,9.167,148.702
C04348=1179.610,416.913,-86.137,-176.018,9.166,148.702
C04349=1179.608,416.682,-86.104,-176.018,9.164,148.701
C04350=1179.608,416.450,-86.072,-176.018,9.162,148.701
C04351=1179.608,416.219,-86.038,-176.018,9.161,148.701
C04352=1179.610,415.987,-86.004,-176.018,9.160,148.700
C04353=1179.612,415.755,-85.970,-176.018,9.157,148.700
C04354=1179.615,415.524,-85.937,-176.018,9.156,148.699
C04355=1179.619,415.292,-85.904,-176.018,9.154,148.699
C04356=1179.624,415.044,-85.868,-176.017,9.152,148.698
C04357=1179.627,414.797,-85.831,-176.017,9.150,148.698
C04358=1179.632,414.549,-85.795,-176.017,9.148,148.697
C04359=1179.635,414.302,-85.760,-176.017,9.147,148.697
C04360=1179.639,414.055,-85.723,-176.017,9.145,148.696
C04361=1179.643,413.807,-85.687,-176.017,9.143,148.695
C04362=1179.647,413.560,-85.652,-176.017,9.141,148.695
C04363=1179.651,413.313,-85.615,-176.017,9.139,148.694
C04364=1179.655,413.066,-85.580,-176.017,9.137,148.694
C04365=1179.659,412.818,-85.544,-176.017,9.134,148.693
C04366=1179.663,412.571,-85.507,-176.016,9.133,148.693
C04367=1179.666,412.324,-85.472,-176.017,9.131,148.692
C04368=1179.671,412.076,-85.436,-176.016,9.129,148.692
C04369=1179.674,411.828,-85.400,-176.016,9.127,148.691
C04370=1179.678,411.581,-85.364,-176.016,9.125,148.691
C04371=1179.682,411.334,-85.328,-176.016,9.123,148.690
C04372=1179.686,411.087,-85.292,-176.015,9.121,148.689
C04373=1179.691,410.840,-85.256,-176.016,9.119,148.689
C04374=1179.694,410.592,-85.220,-176.015,9.117,148.688
C04375=1179.698,410.345,-85.184,-176.015,9.115,148.688
C04376=1179.702,410.097,-85.148,-176.016,9.113,148.687
C04377=1179.706,409.850,-85.112,-176.015,9.111,148.687
C04378=1179.710,409.602,-85.076,-176.015,9.109,148.686
C04379=1179.714,409.355,-85.040,-176.015,9.107,148.686
C04380=1179.717,409.107,-85.005,-176.015,9.105,148.685
C04381=1179.722,408.861,-84.968,-176.015,9.102,148.684
C04382=1179.726,408.613,-84.933,-176.015,9.101,148.684
C04383=1179.729,408.366,-84.897,-176.015,9.099,148.683
C04384=1179.734,408.118,-84.861,-176.015,9.096,148.683
C04385=1179.737,407.871,-84.825,-176.014,9.095,148.682
C04386=1179.741,407.623,-84.789,-176.014,9.092,148.681
C04387=1179.745,407.376,-84.753,-176.015,9.090,148.681
C04388=1179.749,407.128,-84.718,-176.014,9.088,148.680
C04389=1179.753,406.881,-84.681,-176.014,9.086,148.680
C04390=1179.757,406.634,-84.646,-176.014,9.083,148.679
C04391=1179.761,406.387,-84.610,-176.014,9.082,148.679
C04392=1179.765,406.139,-84.574,-176.014,9.079,148.678
C04393=1179.769,405.892,-84.538,-176.014,9.077,148.677
C04394=1179.772,405.644,-84.502,-176.013,9.075,148.677
C04395=1179.777,405.397,-84.466,-176.013,9.073,148.676
C04396=1179.780,405.149,-84.430,-176.014,9.071,148.676
C04397=1179.785,404.902,-84.395,-176.014,9.068,148.675
C04398=1179.789,404.654,-84.359,-176.013,9.067,148.674
C04399=1179.792,404.408,-84.323,-176.013,9.064,148.674
C04400=1179.796,404.160,-84.287,-176.013,9.062,148.673
C04401=1179.800,403.912,-84.251,-176.013,9.060,148.673
C04402=1179.804,403.665,-84.215,-176.013,9.057,148.672
C04403=1179.808,403.417,-84.180,-176.013,9.056,148.672
C04404=1179.812,403.171,-84.143,-176.013,9.053,148.671
C04405=1179.816,402.923,-84.108,-176.013,9.051,148.670
C04406=1179.820,402.676,-84.072,-176.013,9.048,148.670
C04407=1179.824,402.428,-84.036,-176.013,9.046,148.669
C04408=1179.828,402.180,-84.001,-176.012,9.044,148.668
C04409=1179.832,401.933,-83.965,-176.012,9.042,148.668
C04410=1179.835,401.685,-83.930,-176.012,9.039,148.667
C04411=1179.840,401.439,-83.893,-176.012,9.037,148.666
C04412=1179.844,401.191,-83.858,-176.013,9.034,148.666
C04413=1179.847,400.944,-83.822,-176.012,9.032,148.665
C04414=1179.852,400.696,-83.786,-176.013,9.030,148.665
C04415=1179.855,400.449,-83.750,-176.013,9.027,148.664
C04416=1179.859,400.201,-83.715,-176.013,9.025,148.663
C04417=1179.864,399.954,-83.679,-176.013,9.022,148.663
C04418=1179.868,399.707,-83.643,-176.012,9.020,148.662
C04419=1179.871,399.460,-83.607,-176.013,9.017,148.661
C04420=1179.875,399.212,-83.572,-176.013,9.015,148.661
C04421=1179.879,398.964,-83.535,-176.013,9.013,148.660
C04422=1179.883,398.717,-83.500,-176.013,9.010,148.660
C04423=1179.887,398.470,-83.465,-176.012,9.007,148.659
C04424=1179.891,398.223,-83.429,-176.013,9.005,148.658
C04425=1179.895,397.975,-83.393,-176.013,9.003,148.658
C04426=1179.899,397.727,-83.357,-176.013,9.000,148.657
C04427=1179.902,397.480,-83.322,-176.013,8.998,148.656
C04428=1179.907,397.233,-83.286,-176.013,8.996,148.656
C04429=1179.911,396.985,-83.251,-176.013,8.993,148.655
C04430=1179.915,396.738,-83.215,-176.013,8.990,148.654
C04431=1179.918,396.490,-83.180,-176.013,8.988,148.654
C04432=1179.923,396.242,-83.143,-176.013,8.985,148.653
C04433=1179.927,395.996,-83.107,-176.013,8.982,148.653
C04434=1179.930,395.749,-83.072,-176.013,8.980,148.652
C04435=1179.934,395.501,-83.036,-176.013,8.977,148.651
C04436=1179.938,395.254,-83.001,-176.013,8.975,148.651
C04437=1179.942,395.006,-82.965,-176.013,8.972,148.650
C04438=1179.946,394.759,-82.930,-176.014,8.969,148.649
C04439=1179.950,394.512,-82.894,-176.014,8.967,148.649
C04440=1179.954,394.264,-82.858,-176.014,8.964,148.648
C04441=1179.958,394.016,-82.822,-176.014,8.962,148.647
C04442=1179.962,393.769,-82.787,-176.014,8.959,148.647
C04443=1179.966,393.522,-82.752,-176.015,8.956,148.646
C04444=1179.970,393.274,-82.716,-176.014,8.954,148.645
C04445=1179.973,393.027,-82.680,-176.015,8.951,148.645
C04446=1179.978,392.779,-82.644,-176.015,8.948,148.644
C04447=1179.981,392.532,-82.609,-176.015,8.946,148.643
C04448=1179.986,392.248,-82.569,-176.015,8.942,148.643
C04449=1179.990,391.963,-82.528,-176.016,8.939,148.642
C04450=1179.995,391.679,-82.487,-176.017,8.936,148.641
C04451=1180.000,391.394,-82.446,-176.017,8.932,148.640
C04452=1180.004,391.148,-82.411,-176.017,8.930,148.640
C04453=1180.007,390.900,-82.376,-176.018,8.927,148.639
C04454=1180.012,390.652,-82.340,-176.017,8.924,148.638
C04455=1180.016,390.405,-82.304,-176.018,8.921,148.638
C04456=1180.020,390.158,-82.269,-176.018,8.918,148.637
C04457=1180.023,389.911,-82.233,-176.019,8.915,148.636
C04458=1180.027,389.663,-82.198,-176.019,8.913,148.636
C04459=1180.031,389.416,-82.162,-176.020,8.910,148.635
C04460=1180.036,389.168,-82.126,-176.019,8.907,148.634
C04461=1180.040,388.920,-82.092,-176.020,8.904,148.634
C04462=1180.043,388.673,-82.056,-176.021,8.901,148.633
C04463=1180.047,388.425,-82.020,-176.021,8.898,148.633
C04464=1180.051,388.179,-81.985,-176.021,8.895,148.632
C04465=1180.055,387.931,-81.950,-176.022,8.892,148.631
C04466=1180.059,387.684,-81.914,-176.022,8.889,148.630
C04467=1180.062,387.436,-81.879,-176.023,8.886,148.630
C04468=1180.067,387.189,-81.844,-176.024,8.883,148.629
C04469=1180.071,386.941,-81.808,-176.024,8.880,148.629
C04470=1180.075,386.693,-81.773,-176.024,8.877,148.628
C04471=1180.079,386.446,-81.737,-176.025,8.874,148.627
C04472=1180.083,386.199,-81.702,-176.025,8.871,148.627
C04473=1180.087,385.951,-81.667,-176.026,8.868,148.626
C04474=1180.090,385.703,-81.631,-176.027,8.864,148.625
C04475=1180.095,385.457,-81.596,-176.027,8.861,148.625
C04476=1180.098,385.209,-81.561,-176.028,8.858,148.624
C04477=1180.102,384.962,-81.525,-176.029,8.856,148.624
C04478=1180.107,384.714,-81.491,-176.029,8.853,148.623
C04479=1180.110,384.467,-81.455,-176.030,8.849,148.622
C04480=1180.114,384.219,-81.420,-176.031,8.846,148.622
C04481=1180.118,383.971,-81.385,-176.031,8.843,148.621
C04482=1180.122,383.724,-81.350,-176.032,8.840,148.620
C04483=1180.127,383.476,-81.313,-176.033,8.837,148.620
C04484=1180.130,383.229,-81.278,-176.033,8.834,148.619
C04485=1180.135,382.982,-81.243,-176.035,8.830,148.619
C04486=1180.139,382.734,-81.208,-176.036,8.827,148.618
C04487=1180.142,382.487,-81.172,-176.036,8.824,148.617
C04488=1180.147,382.239,-81.138,-176.037,8.820,148.617
C04489=1180.150,381.992,-81.102,-176.038,8.817,148.616
C04490=1180.154,381.744,-81.067,-176.038,8.814,148.615
C04491=1180.159,381.497,-81.032,-176.039,8.811,148.615
C04492=1180.162,381.249,-80.997,-176.040,8.808,148.614
C04493=1180.166,381.002,-80.961,-176.042,8.804,148.614
C04494=1180.171,380.754,-80.927,-176.042,8.801,148.613
C04495=1180.174,380.507,-80.891,-176.043,8.798,148.612
C04496=1180.178,380.259,-80.856,-176.044,8.795,148.612
C04497=1180.182,380.012,-80.821,-176.045,8.791,148.611
C04498=1180.185,379.765,-80.786,-176.046,8.788,148.611
C04499=1180.190,379.517,-80.752,-176.047,8.785,148.610
C04500=1180.194,379.270,-80.716,-176.048,8.781,148.609
C04501=1180.198,379.022,-80.681,-176.049,8.778,148.609
C04502=1180.202,378.775,-80.646,-176.050,8.774,148.608
C04503=1180.206,378.527,-80.611,-176.052,8.771,148.608
C04504=1180.209,378.279,-80.576,-176.053,8.768,148.607
C04505=1180.214,378.032,-80.541,-176.054,8.765,148.607
C04506=1180.218,377.784,-80.506,-176.055,8.761,148.606
C04507=1180.222,377.537,-80.471,-176.056,8.758,148.605
C04508=1180.226,377.289,-80.436,-176.057,8.754,148.605
C04509=1180.230,377.041,-80.401,-176.058,8.751,148.604
C04510=1180.234,376.794,-80.366,-176.060,8.747,148.604
C04511=1180.237,376.547,-80.332,-176.061,8.744,148.603
C04512=1180.242,376.300,-80.296,-176.062,8.740,148.603
C04513=1180.246,376.052,-80.261,-176.063,8.737,148.602
C04514=1180.250,375.804,-80.227,-176.065,8.733,148.602
C04515=1180.254,375.557,-80.191,-176.065,8.730,148.601
C04516=1180.258,375.309,-80.157,-176.067,8.727,148.601
C04517=1180.262,375.062,-80.121,-176.068,8.723,148.600
C04518=1180.265,374.814,-80.087,-176.069,8.720,148.599
C04519=1180.270,374.567,-80.053,-176.071,8.717,148.599
C04520=1180.274,374.319,-80.017,-176.072,8.713,148.598
C04521=1180.278,374.071,-79.982,-176.074,8.709,148.598
C04522=1180.282,373.824,-79.947,-176.075,8.706,148.597
C04523=1180.285,373.576,-79.913,-176.077,8.703,148.597
C04524=1180.290,373.329,-79.878,-176.077,8.699,148.596
C04525=1180.294,373.081,-79.844,-176.079,8.696,148.596
C04526=1180.298,372.834,-79.808,-176.081,8.692,148.595
C04527=1180.302,372.586,-79.774,-176.082,8.689,148.595
C04528=1180.306,372.339,-79.740,-176.083,8.685,148.594
C04529=1180.309,372.091,-79.704,-176.085,8.682,148.594
C04530=1180.314,371.844,-79.670,-176.086,8.678,148.593
C04531=1180.318,371.596,-79.635,-176.088,8.675,148.593
C04532=1180.322,371.349,-79.601,-176.090,8.671,148.592
C04533=1180.325,371.101,-79.566,-176.091,8.667,148.592
C04534=1180.330,370.854,-79.531,-176.092,8.665,148.591
C04535=1180.334,370.606,-79.496,-176.094,8.661,148.591
C04536=1180.338,370.359,-79.462,-176.095,8.657,148.590
C04537=1180.342,370.110,-79.428,-176.097,8.653,148.590
C04538=1180.346,369.864,-79.392,-176.098,8.651,148.589
C04539=1180.349,369.616,-79.358,-176.100,8.647,148.589
C04540=1180.354,369.368,-79.324,-176.102,8.643,148.588
C04541=1180.358,369.120,-79.289,-176.103,8.639,148.588
C04542=1180.362,368.873,-79.255,-176.105,8.636,148.588
C04543=1180.365,368.625,-79.220,-176.107,8.632,148.587
C04544=1180.370,368.378,-79.186,-176.108,8.629,148.587
C04545=1180.373,368.130,-79.151,-176.110,8.625,148.586
C04546=1180.378,367.882,-79.117,-176.112,8.622,148.586
C04547=1180.382,367.634,-79.082,-176.113,8.618,148.585
C04548=1180.385,367.388,-79.048,-176.115,8.615,148.585
C04549=1180.389,367.140,-79.013,-176.117,8.611,148.584
C04550=1180.394,366.892,-78.978,-176.119,8.607,148.584
C04551=1180.398,366.645,-78.944,-176.120,8.605,148.584
C04552=1180.403,366.363,-78.906,-176.123,8.600,148.583
C04553=1180.406,366.081,-78.866,-176.124,8.597,148.583
C04554=1180.411,365.799,-78.827,-176.127,8.592,148.582
C04555=1180.415,365.518,-78.788,-176.129,8.588,148.582
C04556=1180.420,365.270,-78.754,-176.130,8.585,148.581
C04557=1180.424,365.023,-78.720,-176.132,8.581,148.581
C04558=1180.428,364.775,-78.685,-176.134,8.578,148.580
C04559=1180.432,364.528,-78.651,-176.136,8.574,148.580
C04560=1180.436,364.280,-78.616,-176.138,8.570,148.580
C04561=1180.439,364.033,-78.582,-176.139,8.567,148.579
C04562=1180.444,363.785,-78.549,-176.142,8.563,148.579
C04563=1180.448,363.537,-78.514,-176.144,8.560,148.578
C04564=1180.452,363.290,-78.480,-176.145,8.556,148.578
C04565=1180.455,363.042,-78.446,-176.147,8.553,148.578
C04566=1180.460,362.794,-78.411,-176.149,8.549,148.577
C04567=1180.464,362.547,-78.377,-176.151,8.546,148.577
C04568=1180.468,362.299,-78.343,-176.153,8.542,148.577
C04569=1180.472,362.051,-78.309,-176.155,8.538,148.576
C04570=1180.476,361.804,-78.275,-176.157,8.535,148.576
C04571=1180.480,361.556,-78.241,-176.159,8.531,148.575
C04572=1180.484,361.309,-78.206,-176.161,8.528,148.575
C04573=1180.488,361.061,-78.173,-176.163,8.525,148.575
C04574=1180.492,360.813,-78.138,-176.165,8.521,148.574
C04575=1180.496,360.566,-78.104,-176.167,8.518,148.574
C04576=1180.500,360.318,-78.071,-176.169,8.514,148.574
C04577=1180.504,360.070,-78.036,-176.171,8.511,148.573
C04578=1180.508,359.823,-78.002,-176.173,8.507,148.573
C04579=1180.512,359.575,-77.969,-176.175,8.504,148.573
C04580=1180.516,359.327,-77.934,-176.177,8.500,148.572
C04581=1180.520,359.080,-77.901,-176.179,8.497,148.572
C04582=1180.525,358.832,-77.867,-176.181,8.493,148.572
C04583=1180.528,358.584,-77.833,-176.184,8.490,148.572
C04584=1180.532,358.337,-77.799,-176.186,8.485,148.571
C04585=1180.537,358.089,-77.765,-176.188,8.482,148.571
C04586=1180.541,357.842,-77.731,-176.190,8.478,148.570
C04587=1180.544,357.593,-77.698,-176.192,8.475,148.570
C04588=1180.549,357.346,-77.663,-176.194,8.472,148.570
C04589=1180.553,357.098,-77.630,-176.196,8.468,148.570
C04590=1180.557,356.851,-77.596,-176.199,8.465,148.569
C04591=1180.560,356.603,-77.563,-176.200,8.461,148.569
C04592=1180.565,356.355,-77.528,-176.203,8.458,148.569
C04593=1180.569,356.108,-77.495,-176.205,8.455,148.568
C04594=1180.573,355.860,-77.461,-176.207,8.451,148.568
C04595=1180.577,355.612,-77.427,-176.209,8.448,148.568
C04596=1180.581,355.365,-77.393,-176.212,8.444,148.567
C04597=1180.585,355.117,-77.360,-176.214,8.440,148.567
C04598=1180.589,354.870,-77.326,-176.216,8.437,148.567
C04599=1180.594,354.622,-77.292,-176.218,8.433,148.567
C04600=1180.597,354.373,-77.259,-176.220,8.430,148.566
C04601=1180.601,354.126,-77.225,-176.222,8.426,148.566
C04602=1180.605,353.878,-77.192,-176.225,8.423,148.566
C04603=1180.609,353.631,-77.158,-176.227,8.420,148.566
C04604=1180.614,353.383,-77.124,-176.229,8.416,148.565
C04605=1180.618,353.135,-77.091,-176.231,8.413,148.565
C04606=1180.622,352.887,-77.057,-176.233,8.410,148.565
C04607=1180.626,352.640,-77.024,-176.235,8.406,148.564
C04608=1180.630,352.392,-76.990,-176.238,8.403,148.564
C04609=1180.634,352.145,-76.957,-176.240,8.399,148.564
C04610=1180.638,351.897,-76.923,-176.242,8.395,148.564
C04611=1180.643,351.649,-76.890,-176.245,8.392,148.563
C04612=1180.646,351.401,-76.856,-176.247,8.389,148.563
C04613=1180.650,351.153,-76.823,-176.249,8.385,148.563
C04614=1180.654,350.906,-76.789,-176.251,8.382,148.562
C04615=1180.658,350.658,-76.756,-176.253,8.378,148.562
C04616=1180.662,350.411,-76.723,-176.255,8.375,148.562
C04617=1180.666,350.163,-76.690,-176.258,8.372,148.562
C04618=1180.671,349.915,-76.656,-176.260,8.368,148.562
C04619=1180.675,349.667,-76.623,-176.262,8.365,148.561
C04620=1180.678,349.419,-76.590,-176.265,8.362,148.561
C04621=1180.683,349.172,-76.555,-176.267,8.358,148.561
C04622=1180.687,348.924,-76.522,-176.269,8.355,148.560
C04623=1180.691,348.676,-76.489,-176.271,8.352,148.560
C04624=1180.695,348.428,-76.456,-176.273,8.348,148.560
C04625=1180.699,348.181,-76.423,-176.275,8.345,148.560
C04626=1180.704,347.933,-76.390,-176.278,8.342,148.560
C04627=1180.708,347.685,-76.356,-176.281,8.337,148.559
C04628=1180.712,347.438,-76.323,-176.283,8.334,148.559
C04629=1180.716,347.190,-76.290,-176.285,8.331,148.559
C04630=1180.720,346.942,-76.257,-176.287,8.328,148.559
C04631=1180.724,346.694,-76.224,-176.290,8.324,148.558
C04632=1180.728,346.447,-76.191,-176.292,8.321,148.558
C04633=1180.732,346.199,-76.157,-176.294,8.318,148.558
C04634=1180.737,345.951,-76.124,-176.296,8.314,148.558
C04635=1180.740,345.704,-76.092,-176.299,8.311,148.558
C04636=1180.744,345.456,-76.059,-176.301,8.308,148.557
C04637=1180.748,345.208,-76.025,-176.303,8.304,148.557
C04638=1180.752,344.961,-75.992,-176.305,8.301,148.557
C04639=1180.757,344.712,-75.960,-176.308,8.298,148.557
C04640=1180.761,344.464,-75.927,-176.310,8.294,148.557
C04641=1180.765,344.217,-75.893,-176.312,8.291,148.556
C04642=1180.769,343.969,-75.860,-176.314,8.288,148.556
C04643=1180.773,343.721,-75.827,-176.317,8.284,148.556
C04644=1180.778,343.474,-75.794,-176.319,8.281,148.556
C04645=1180.781,343.226,-75.762,-176.321,8.278,148.555
C04646=1180.785,342.978,-75.729,-176.324,8.275,148.555
C04647=1180.790,342.730,-75.696,-176.326,8.271,148.555
C04648=1180.794,342.482,-75.663,-176.328,8.268,148.555
C04649=1180.798,342.234,-75.630,-176.331,8.265,148.555
C04650=1180.802,341.986,-75.597,-176.333,8.262,148.555
C04651=1180.806,341.739,-75.565,-176.335,8.258,148.554
C04652=1180.810,341.491,-75.531,-176.338,8.255,148.554
C04653=1180.814,341.243,-75.499,-176.340,8.252,148.554
C04654=1180.818,340.995,-75.466,-176.342,8.248,148.554
C04655=1180.823,340.747,-75.433,-176.344,8.245,148.554
C04656=1180.827,340.469,-75.396,-176.348,8.241,148.553
C04657=1180.832,340.189,-75.360,-176.350,8.237,148.553
C04658=1180.836,339.910,-75.323,-176.353,8.234,148.553
C04659=1180.841,339.631,-75.286,-176.356,8.230,148.553
C04660=1180.845,339.384,-75.253,-176.358,8.226,148.552
C04661=1180.849,339.135,-75.221,-176.360,8.223,148.552
C04662=1180.854,338.888,-75.187,-176.363,8.220,148.552
C04663=1180.857,338.640,-75.156,-176.365,8.217,148.552
C04664=1180.862,338.393,-75.123,-176.367,8.213,148.552
C04665=1180.866,338.144,-75.090,-176.370,8.210,148.552
C04666=1180.870,337.897,-75.058,-176.372,8.207,148.551
C04667=1180.874,337.648,-75.025,-176.375,8.204,148.551
C04668=1180.878,337.401,-74.992,-176.377,8.200,148.551
C04669=1180.882,337.153,-74.960,-176.379,8.197,148.551
C04670=1180.886,336.905,-74.927,-176.381,8.194,148.551
C04671=1180.891,336.657,-74.895,-176.384,8.191,148.551
C04672=1180.895,336.410,-74.863,-176.386,8.187,148.551
C04673=1180.899,336.161,-74.830,-176.389,8.184,148.550
C04674=1180.903,335.914,-74.798,-176.391,8.181,148.550
C04675=1180.907,335.666,-74.765,-176.394,8.178,148.550
C04676=1180.911,335.417,-74.733,-176.396,8.175,148.550
C04677=1180.915,335.170,-74.700,-176.398,8.171,148.550
C04678=1180.920,334.922,-74.668,-176.400,8.168,148.550
C04679=1180.923,334.675,-74.635,-176.403,8.165,148.550
C04680=1180.928,334.427,-74.603,-176.405,8.162,148.549
C04681=1180.931,334.178,-74.571,-176.408,8.158,148.549
C04682=1180.936,333.931,-74.538,-176.410,8.155,148.549
C04683=1180.940,333.683,-74.507,-176.413,8.152,148.549
C04684=1180.944,333.435,-74.474,-176.415,8.149,148.549
C04685=1180.948,333.187,-74.442,-176.417,8.145,148.548
C04686=1180.952,332.939,-74.409,-176.420,8.142,148.548
C04687=1180.957,332.692,-74.377,-176.422,8.139,148.548
C04688=1180.961,332.444,-74.345,-176.424,8.136,148.548
C04689=1180.965,332.196,-74.313,-176.427,8.133,148.548
C04690=1180.969,331.948,-74.280,-176.429,8.129,148.548
C04691=1180.973,331.701,-74.249,-176.432,8.126,148.548
C04692=1180.977,331.452,-74.216,-176.434,8.123,148.548
C04693=1180.981,331.204,-74.184,-176.437,8.120,148.547
C04694=1180.986,330.956,-74.152,-176.439,8.117,148.547
C04695=1180.990,330.708,-74.120,-176.441,8.113,148.547
C04696=1180.994,330.460,-74.088,-176.443,8.111,148.547
C04697=1180.998,330.213,-74.055,-176.446,8.108,148.547
C04698=1181.002,329.965,-74.024,-176.448,8.105,148.547
C04699=1181.007,329.717,-73.992,-176.450,8.101,148.547
C04700=1181.010,329.469,-73.960,-176.453,8.098,148.547
C04701=1181.015,329.221,-73.927,-176.455,8.095,148.546
C04702=1181.019,328.973,-73.896,-176.458,8.092,148.546
C04703=1181.023,328.725,-73.864,-176.460,8.089,148.546
C04704=1181.027,328.477,-73.831,-176.463,8.085,148.546
C04705=1181.031,328.230,-73.800,-176.465,8.082,148.546
C04706=1181.035,327.982,-73.768,-176.468,8.079,148.546
C04707=1181.040,327.733,-73.736,-176.470,8.076,148.546
C04708=1181.044,327.486,-73.704,-176.473,8.073,148.546
C04709=1181.048,327.238,-73.672,-176.475,8.070,148.546
C04710=1181.052,326.989,-73.640,-176.478,8.066,148.545
C04711=1181.056,326.742,-73.608,-176.480,8.063,148.545
C04712=1181.060,326.494,-73.577,-176.483,8.060,148.545
C04713=1181.065,326.246,-73.544,-176.485,8.057,148.545
C04714=1181.069,325.998,-73.513,-176.488,8.054,148.545
C04715=1181.073,325.750,-73.482,-176.490,8.051,148.545
C04716=1181.077,325.502,-73.450,-176.493,8.048,148.545
C04717=1181.082,325.254,-73.418,-176.495,8.044,148.545
C04718=1181.085,325.006,-73.386,-176.497,8.041,148.545
C04719=1181.090,324.759,-73.354,-176.500,8.038,148.544
C04720=1181.093,324.511,-73.322,-176.502,8.035,148.544
C04721=1181.098,324.262,-73.291,-176.505,8.032,148.544
C04722=1181.102,324.014,-73.259,-176.507,8.029,148.544
C04723=1181.106,323.766,-73.227,-176.510,8.025,148.544
C04724=1181.110,323.519,-73.196,-176.512,8.022,148.544
C04725=1181.114,323.270,-73.165,-176.515,8.019,148.544
C04726=1181.118,323.022,-73.133,-176.517,8.017,148.544
C04727=1181.123,322.775,-73.101,-176.519,8.013,148.544
C04728=1181.127,322.527,-73.069,-176.522,8.010,148.544
C04729=1181.131,322.279,-73.038,-176.524,8.007,148.543
C04730=1181.135,322.031,-73.006,-176.527,8.004,148.543
C04731=1181.139,321.783,-72.975,-176.529,8.001,148.543
C04732=1181.143,321.535,-72.944,-176.532,7.998,148.543
C04733=1181.148,321.287,-72.912,-176.534,7.995,148.543
C04734=1181.152,321.039,-72.880,-176.537,7.992,148.543
C04735=1181.156,320.790,-72.849,-176.539,7.988,148.543
C04736=1181.161,320.543,-72.817,-176.542,7.985,148.543
C04737=1181.165,320.294,-72.786,-176.544,7.982,148.543
C04738=1181.169,320.047,-72.755,-176.547,7.979,148.543
C04739=1181.173,319.798,-72.724,-176.549,7.976,148.542
C04740=1181.177,319.551,-72.692,-176.552,7.973,148.542
C04741=1181.181,319.303,-72.660,-176.554,7.970,148.542
C04742=1181.186,319.055,-72.629,-176.557,7.966,148.542
C04743=1181.189,318.807,-72.598,-176.559,7.963,148.542
C04744=1181.194,318.559,-72.567,-176.561,7.961,148.542
C04745=1181.198,318.311,-72.535,-176.564,7.958,148.542
C04746=1181.202,318.063,-72.504,-176.566,7.955,148.542
C04747=1181.206,317.814,-72.473,-176.569,7.952,148.542
C04748=1181.210,317.567,-72.442,-176.572,7.949,148.542
C04749=1181.215,317.319,-72.411,-176.574,7.945,148.542
C04750=1181.219,317.071,-72.379,-176.576,7.942,148.542
C04751=1181.223,316.823,-72.348,-176.579,7.939,148.542
C04752=1181.227,316.575,-72.316,-176.581,7.936,148.542
C04753=1181.232,316.327,-72.286,-176.584,7.933,148.542
C04754=1181.236,316.078,-72.255,-176.586,7.930,148.541
C04755=1181.240,315.831,-72.223,-176.589,7.927,148.541
C04756=1181.244,315.582,-72.192,-176.592,7.924,148.541
C04757=1181.249,315.334,-72.161,-176.594,7.921,148.541
C04758=1181.253,315.087,-72.130,-176.596,7.918,148.541
C04759=1181.256,314.839,-72.099,-176.599,7.915,148.541
C04760=1181.261,314.562,-72.064,-176.602,7.911,148.541
C04761=1181.266,314.285,-72.030,-176.605,7.908,148.541
C04762=1181.271,314.009,-71.995,-176.607,7.905,148.541
C04763=1181.275,313.732,-71.960,-176.610,7.901,148.541
C04764=1181.280,313.484,-71.930,-176.613,7.898,148.541
C04765=1181.284,313.235,-71.899,-176.616,7.895,148.541
C04766=1181.289,312.987,-71.868,-176.618,7.892,148.541
C04767=1181.292,312.740,-71.837,-176.620,7.889,148.541
C04768=1181.296,312.492,-71.806,-176.623,7.886,148.541
C04769=1181.301,312.244,-71.775,-176.625,7.883,148.541
C04770=1181.305,311.995,-71.744,-176.628,7.880,148.541
C04771=1181.309,311.747,-71.713,-176.630,7.877,148.541
C04772=1181.313,311.500,-71.683,-176.633,7.874,148.540
C04773=1181.317,311.251,-71.652,-176.635,7.871,148.540
C04774=1181.322,311.003,-71.621,-176.638,7.868,148.540
C04775=1181.326,310.756,-71.590,-176.640,7.864,148.540
C04776=1181.330,310.507,-71.558,-176.643,7.861,148.540
C04777=1181.334,310.259,-71.528,-176.645,7.859,148.540
C04778=1181.339,310.011,-71.498,-176.647,7.856,148.540
C04779=1181.343,309.763,-71.467,-176.650,7.853,148.540
C04780=1181.347,309.515,-71.436,-176.653,7.850,148.540
C04781=1181.351,309.267,-71.405,-176.655,7.847,148.540
C04782=1181.356,309.019,-71.375,-176.658,7.844,148.540
C04783=1181.360,308.770,-71.344,-176.661,7.841,148.540
C04784=1181.364,308.523,-71.313,-176.663,7.838,148.540
C04785=1181.368,308.275,-71.283,-176.666,7.834,148.540
C04786=1181.373,308.027,-71.252,-176.668,7.831,148.540
C04787=1181.377,307.778,-71.222,-176.670,7.829,148.540
C04788=1181.381,307.530,-71.191,-176.673,7.826,148.540
C04789=1181.386,307.282,-71.161,-176.675,7.823,148.540
C04790=1181.390,307.034,-71.130,-176.678,7.820,148.540
C04791=1181.394,306.786,-71.099,-176.681,7.817,148.540
C04792=1181.398,306.538,-71.068,-176.683,7.814,148.540
C04793=1181.402,306.290,-71.038,-176.686,7.811,148.540
C04794=1181.407,306.042,-71.008,-176.689,7.808,148.540
C04795=1181.410,305.793,-70.978,-176.691,7.805,148.540
C04796=1181.415,305.545,-70.947,-176.693,7.802,148.539
C04797=1181.420,305.297,-70.916,-176.696,7.799,148.539
C04798=1181.423,305.050,-70.886,-176.698,7.796,148.539
C04799=1181.428,304.801,-70.856,-176.701,7.793,148.539
C04800=1181.432,304.553,-70.825,-176.703,7.790,148.539
C04801=1181.436,304.305,-70.795,-176.706,7.787,148.539
C04802=1181.440,304.057,-70.765,-176.709,7.784,148.539
C04803=1181.445,303.809,-70.734,-176.711,7.782,148.539
C04804=1181.449,303.561,-70.704,-176.713,7.778,148.539
C04805=1181.454,303.313,-70.674,-176.716,7.775,148.539
C04806=1181.458,303.064,-70.643,-176.719,7.772,148.539
C04807=1181.462,302.816,-70.613,-176.721,7.769,148.539
C04808=1181.466,302.568,-70.582,-176.724,7.766,148.539
C04809=1181.471,302.320,-70.553,-176.726,7.763,148.539
C04810=1181.475,302.072,-70.522,-176.729,7.761,148.539
C04811=1181.479,301.824,-70.492,-176.731,7.758,148.539
C04812=1181.483,301.576,-70.462,-176.734,7.755,148.539
C04813=1181.487,301.327,-70.431,-176.736,7.752,148.539
C04814=1181.491,301.079,-70.402,-176.739,7.749,148.539
C04815=1181.496,300.831,-70.371,-176.742,7.746,148.539
C04816=1181.500,300.583,-70.342,-176.744,7.743,148.539
C04817=1181.505,300.335,-70.311,-176.747,7.741,148.539
C04818=1181.509,300.087,-70.281,-176.749,7.737,148.539
C04819=1181.513,299.839,-70.251,-176.752,7.734,148.539
C04820=1181.518,299.590,-70.221,-176.754,7.731,148.539
C04821=1181.522,299.343,-70.191,-176.757,7.728,148.539
C04822=1181.526,299.093,-70.161,-176.760,7.725,148.539
C04823=1181.530,298.846,-70.130,-176.762,7.722,148.539
C04824=1181.534,298.597,-70.101,-176.764,7.720,148.539
C04825=1181.539,298.349,-70.070,-176.767,7.717,148.539
C04826=1181.543,298.101,-70.041,-176.770,7.714,148.539
C04827=1181.547,297.854,-70.011,-176.772,7.711,148.539
C04828=1181.552,297.605,-69.980,-176.775,7.708,148.539
C04829=1181.556,297.357,-69.951,-176.777,7.704,148.539
C04830=1181.560,297.109,-69.921,-176.780,7.702,148.539
C04831=1181.564,296.861,-69.891,-176.782,7.699,148.539
C04832=1181.569,296.612,-69.861,-176.785,7.696,148.539
C04833=1181.573,296.365,-69.831,-176.788,7.693,148.539
C04834=1181.577,296.116,-69.802,-176.790,7.690,148.539
C04835=1181.582,295.868,-69.772,-176.793,7.687,148.539
C04836=1181.586,295.620,-69.742,-176.795,7.685,148.539
C04837=1181.590,295.372,-69.712,-176.798,7.682,148.539
C04838=1181.594,295.124,-69.683,-176.800,7.679,148.539
C04839=1181.598,294.875,-69.653,-176.803,7.676,148.539
C04840=1181.603,294.627,-69.622,-176.806,7.673,148.539
C04841=1181.607,294.379,-69.593,-176.808,7.670,148.539
C04842=1181.611,294.131,-69.563,-176.811,7.668,148.539
C04843=1181.615,293.883,-69.534,-176.813,7.664,148.539
C04844=1181.620,293.634,-69.505,-176.816,7.661,148.539
C04845=1181.624,293.386,-69.474,-176.818,7.658,148.539
C04846=1181.628,293.138,-69.444,-176.821,7.655,148.539
C04847=1181.632,292.890,-69.415,-176.823,7.653,148.539
C04848=1181.637,292.642,-69.385,-176.826,7.650,148.539
C04849=1181.641,292.393,-69.356,-176.829,7.647,148.539
C04850=1181.645,292.145,-69.327,-176.831,7.644,148.539
C04851=1181.649,291.897,-69.297,-176.834,7.641,148.539
C04852=1181.654,291.648,-69.267,-176.836,7.638,148.539
C04853=1181.658,291.400,-69.238,-176.839,7.636,148.539
C04854=1181.662,291.152,-69.207,-176.841,7.633,148.539
C04855=1181.666,290.904,-69.178,-176.844,7.630,148.539
C04856=1181.671,290.656,-69.149,-176.847,7.627,148.539
C04857=1181.675,290.408,-69.119,-176.849,7.624,148.539
C04858=1181.680,290.160,-69.090,-176.852,7.622,148.539
C04859=1181.684,289.912,-69.061,-176.854,7.619,148.539
C04860=1181.688,289.663,-69.031,-176.857,7.616,148.539
C04861=1181.692,289.414,-69.002,-176.860,7.613,148.539
C04862=1181.697,289.166,-68.973,-176.862,7.610,148.539
C04863=1181.701,288.918,-68.943,-176.864,7.607,148.539
C04864=1181.706,288.644,-68.910,-176.867,7.604,148.539
C04865=1181.710,288.369,-68.878,-176.871,7.601,148.539
C04866=1181.715,288.095,-68.846,-176.873,7.598,148.540
C04867=1181.720,287.819,-68.813,-176.876,7.595,148.540
C04868=1181.724,287.571,-68.784,-176.879,7.592,148.540
C04869=1181.728,287.323,-68.755,-176.881,7.589,148.539
C04870=1181.732,287.075,-68.725,-176.883,7.586,148.539
C04871=1181.737,286.827,-68.697,-176.886,7.583,148.539
C04872=1181.741,286.578,-68.667,-176.889,7.580,148.540
C04873=1181.746,286.330,-68.638,-176.891,7.577,148.540
C04874=1181.750,286.082,-68.608,-176.894,7.574,148.540
C04875=1181.754,285.834,-68.579,-176.896,7.572,148.540
C04876=1181.759,285.585,-68.551,-176.899,7.569,148.540
C04877=1181.763,285.337,-68.521,-176.902,7.566,148.540
C04878=1181.767,285.089,-68.492,-176.905,7.563,148.540
C04879=1181.772,284.841,-68.462,-176.907,7.561,148.540
C04880=1181.776,284.592,-68.433,-176.909,7.558,148.540
C04881=1181.781,284.344,-68.404,-176.912,7.555,148.540
C04882=1181.784,284.096,-68.376,-176.915,7.552,148.540
C04883=1181.789,283.847,-68.347,-176.917,7.550,148.540
C04884=1181.793,283.599,-68.317,-176.920,7.547,148.540
C04885=1181.798,283.351,-68.288,-176.922,7.544,148.540
C04886=1181.802,283.103,-68.260,-176.925,7.541,148.540
C04887=1181.806,282.854,-68.230,-176.928,7.538,148.540
C04888=1181.810,282.606,-68.202,-176.930,7.536,148.540
C04889=1181.815,282.358,-68.173,-176.933,7.533,148.540
C04890=1181.819,282.110,-68.143,-176.936,7.530,148.540
C04891=1181.824,281.861,-68.115,-176.938,7.527,148.540
C04892=1181.828,281.613,-68.085,-176.940,7.525,148.540
C04893=1181.832,281.365,-68.057,-176.943,7.522,148.540
C04894=1181.836,281.117,-68.028,-176.946,7.519,148.540
C04895=1181.841,280.868,-67.999,-176.949,7.516,148.541
C04896=1181.845,280.619,-67.970,-176.951,7.514,148.541
C04897=1181.849,280.372,-67.942,-176.953,7.511,148.541
C04898=1181.854,280.123,-67.913,-176.956,7.508,148.541
C04899=1181.858,279.874,-67.884,-176.958,7.506,148.541
C04900=1181.863,279.627,-67.855,-176.961,7.503,148.541
C04901=1181.867,279.378,-67.827,-176.964,7.500,148.541
C04902=1181.871,279.130,-67.797,-176.967,7.497,148.541
C04903=1181.876,278.882,-67.769,-176.969,7.494,148.541
C04904=1181.880,278.633,-67.741,-176.971,7.491,148.541
C04905=1181.884,278.385,-67.711,-176.974,7.488,148.541
C04906=1181.889,278.137,-67.683,-176.977,7.485,148.541
C04907=1181.892,277.889,-67.654,-176.979,7.483,148.541
C04908=1181.897,277.640,-67.625,-176.982,7.480,148.541
C04909=1181.902,277.392,-67.597,-176.985,7.477,148.541
C04910=1181.905,277.144,-67.568,-176.987,7.474,148.541
C04911=1181.910,276.895,-67.539,-176.989,7.472,148.541
C04912=1181.915,276.647,-67.511,-176.992,7.469,148.541
C04913=1181.919,276.398,-67.483,-176.995,7.466,148.541
C04914=1181.923,276.150,-67.453,-176.997,7.464,148.542
C04915=1181.927,275.902,-67.425,-177.000,7.461,148.542
C04916=1181.932,275.653,-67.397,-177.002,7.458,148.542
C04917=1181.936,275.405,-67.369,-177.005,7.455,148.542
C04918=1181.940,275.157,-67.340,-177.007,7.453,148.542
C04919=1181.945,274.908,-67.311,-177.011,7.450,148.542
C04920=1181.949,274.660,-67.283,-177.013,7.447,148.542
C04921=1181.954,274.411,-67.254,-177.015,7.445,148.542
C04922=1181.958,274.163,-67.226,-177.018,7.442,148.542
C04923=1181.962,273.915,-67.197,-177.021,7.439,148.542
C04924=1181.966,273.667,-67.169,-177.024,7.436,148.542
C04925=1181.971,273.418,-67.141,-177.026,7.434,148.542
C04926=1181.975,273.170,-67.112,-177.029,7.431,148.542
C04927=1181.980,272.922,-67.084,-177.031,7.428,148.542
C04928=1181.983,272.673,-67.056,-177.033,7.426,148.542
C04929=1181.989,272.425,-67.027,-177.036,7.423,148.543
C04930=1181.992,272.176,-66.999,-177.039,7.420,148.543
C04931=1181.997,271.928,-66.971,-177.041,7.418,148.543
C04932=1182.001,271.680,-66.942,-177.044,7.415,148.543
C04933=1182.006,271.432,-66.914,-177.047,7.412,148.543
C04934=1182.010,271.183,-66.886,-177.049,7.410,148.543
C04935=1182.014,270.936,-66.858,-177.052,7.407,148.543
C04936=1182.019,270.687,-66.829,-177.055,7.404,148.543
C04937=1182.023,270.439,-66.801,-177.057,7.402,148.543
C04938=1182.027,270.190,-66.773,-177.060,7.399,148.543
C04939=1182.032,269.941,-66.746,-177.062,7.396,148.543
C04940=1182.036,269.693,-66.717,-177.065,7.393,148.543
C04941=1182.041,269.445,-66.689,-177.067,7.391,148.543
C04942=1182.045,269.196,-66.661,-177.070,7.388,148.544
C04943=1182.050,268.948,-66.632,-177.073,7.385,148.544
C04944=1182.053,268.699,-66.604,-177.075,7.383,148.544
C04945=1182.058,268.451,-66.577,-177.078,7.380,148.544
C04946=1182.062,268.203,-66.548,-177.081,7.377,148.544
C04947=1182.067,267.955,-66.520,-177.083,7.375,148.544
C04948=1182.070,267.706,-66.492,-177.086,7.372,148.544
C04949=1182.076,267.457,-66.464,-177.088,7.369,148.544
C04950=1182.080,267.209,-66.436,-177.091,7.367,148.544
C04951=1182.084,266.961,-66.408,-177.094,7.364,148.544
C04952=1182.088,266.713,-66.381,-177.096,7.361,148.544
C04953=1182.093,266.464,-66.352,-177.099,7.359,148.545
C04954=1182.097,266.216,-66.325,-177.101,7.356,148.545
C04955=1182.101,265.967,-66.297,-177.103,7.354,148.545
C04956=1182.106,265.719,-66.268,-177.106,7.351,148.545
C04957=1182.111,265.471,-66.240,-177.109,7.348,148.545
C04958=1182.115,265.222,-66.213,-177.112,7.346,148.545
C04959=1182.119,264.974,-66.185,-177.114,7.343,148.545
C04960=1182.123,264.725,-66.157,-177.117,7.340,148.545
C04961=1182.128,264.476,-66.129,-177.119,7.338,148.545
C04962=1182.132,264.229,-66.102,-177.122,7.335,148.545
C04963=1182.136,263.980,-66.074,-177.125,7.332,148.546
C04964=1182.141,263.732,-66.046,-177.127,7.330,148.546
C04965=1182.146,263.483,-66.018,-177.130,7.327,148.546
C04966=1182.150,263.234,-65.991,-177.133,7.324,148.546
C04967=1182.154,262.986,-65.963,-177.135,7.322,148.546
C04968=1182.159,262.713,-65.932,-177.138,7.319,148.546
C04969=1182.164,262.440,-65.902,-177.141,7.316,148.546
C04970=1182.168,262.167,-65.872,-177.144,7.313,148.546
C04971=1182.173,261.895,-65.842,-177.146,7.310,148.546
C04972=1182.177,261.646,-65.813,-177.150,7.308,148.547
C04973=1182.182,261.398,-65.786,-177.152,7.306,148.547
C04974=1182.187,261.149,-65.758,-177.154,7.303,148.547
C04975=1182.191,260.900,-65.730,-177.157,7.300,148.547
C04976=1182.195,260.652,-65.703,-177.159,7.297,148.547
C04977=1182.200,260.404,-65.676,-177.163,7.295,148.547
C04978=1182.204,260.155,-65.648,-177.165,7.293,148.547
C04979=1182.208,259.907,-65.620,-177.167,7.290,148.547
C04980=1182.213,259.658,-65.593,-177.170,7.287,148.547
C04981=1182.217,259.410,-65.566,-177.173,7.285,148.548
C04982=1182.222,259.161,-65.538,-177.176,7.282,148.548
C04983=1182.226,258.913,-65.510,-177.178,7.280,148.548
C04984=1182.231,258.665,-65.483,-177.180,7.277,148.548
C04985=1182.235,258.416,-65.456,-177.183,7.274,148.548
C04986=1182.239,258.168,-65.428,-177.186,7.272,148.548
C04987=1182.244,257.919,-65.401,-177.189,7.269,148.548
C04988=1182.248,257.671,-65.373,-177.191,7.267,148.548
C04989=1182.253,257.423,-65.346,-177.193,7.264,148.548
C04990=1182.257,257.174,-65.319,-177.197,7.261,148.549
C04991=1182.261,256.925,-65.292,-177.199,7.259,148.549
C04992=1182.266,256.677,-65.264,-177.202,7.256,148.549
C04993=1182.270,256.429,-65.237,-177.204,7.254,148.549
C04994=1182.274,256.180,-65.209,-177.207,7.251,148.549
C04995=1182.279,255.932,-65.182,-177.210,7.248,148.549
C04996=1182.283,255.683,-65.155,-177.212,7.246,148.549
C04997=1182.288,255.435,-65.128,-177.215,7.243,148.549
C04998=1182.293,255.186,-65.101,-177.217,7.241,148.550
C04999=1182.297,254.937,-65.073,-177.220,7.238,148.550
C05000=1182.300,254.690,-65.046,-177.222,7.236,148.550
C05001=1182.305,254.441,-65.019,-177.225,7.233,148.550
C05002=1182.310,254.193,-64.992,-177.228,7.230,148.550
C05003=1182.314,253.944,-64.965,-177.230,7.228,148.550
C05004=1182.318,253.695,-64.937,-177.233,7.225,148.550
C05005=1182.323,253.446,-64.910,-177.235,7.223,148.550
C05006=1182.328,253.198,-64.883,-177.238,7.221,148.551
C05007=1182.331,252.950,-64.856,-177.241,7.218,148.551
C05008=1182.336,252.702,-64.829,-177.243,7.215,148.551
C05009=1182.341,252.453,-64.802,-177.246,7.213,148.551
C05010=1182.345,252.205,-64.775,-177.249,7.211,148.551
C05011=1182.349,251.956,-64.747,-177.251,7.208,148.551
C05012=1182.353,251.707,-64.721,-177.254,7.205,148.551
C05013=1182.358,251.459,-64.694,-177.257,7.203,148.552
C05014=1182.363,251.210,-64.667,-177.259,7.201,148.552
C05015=1182.367,250.962,-64.640,-177.262,7.198,148.552
C05016=1182.372,250.713,-64.613,-177.264,7.196,148.552
C05017=1182.376,250.465,-64.586,-177.267,7.193,148.552
C05018=1182.380,250.217,-64.559,-177.269,7.191,148.552
C05019=1182.385,249.968,-64.532,-177.272,7.188,148.553
C05020=1182.389,249.719,-64.505,-177.275,7.185,148.553
C05021=1182.393,249.471,-64.478,-177.277,7.183,148.553
C05022=1182.398,249.222,-64.451,-177.281,7.180,148.553
C05023=1182.403,248.973,-64.425,-177.283,7.178,148.553
C05024=1182.407,248.725,-64.398,-177.285,7.175,148.553
C05025=1182.411,248.477,-64.371,-177.288,7.173,148.553
C05026=1182.416,248.228,-64.344,-177.291,7.170,148.553
C05027=1182.420,247.980,-64.318,-177.293,7.168,148.554
C05028=1182.425,247.731,-64.291,-177.296,7.166,148.554
C05029=1182.429,247.483,-64.264,-177.298,7.163,148.554
C05030=1182.433,247.234,-64.238,-177.301,7.160,148.554
C05031=1182.438,246.986,-64.211,-177.304,7.159,148.554
C05032=1182.443,246.737,-64.184,-177.306,7.156,148.554
C05033=1182.447,246.489,-64.157,-177.309,7.154,148.555
C05034=1182.451,246.240,-64.130,-177.312,7.151,148.555
C05035=1182.456,245.991,-64.104,-177.314,7.149,148.555
C05036=1182.460,245.743,-64.077,-177.317,7.146,148.555
C05037=1182.465,245.495,-64.050,-177.319,7.144,148.555
C05038=1182.469,245.246,-64.025,-177.322,7.141,148.555
C05039=1182.474,244.997,-63.998,-177.324,7.139,148.555
C05040=1182.478,244.749,-63.971,-177.328,7.136,148.556
C05041=1182.482,244.501,-63.944,-177.330,7.134,148.556
C05042=1182.487,244.252,-63.918,-177.333,7.131,148.556
C05043=1182.491,244.003,-63.891,-177.335,7.129,148.556
C05044=1182.496,243.755,-63.864,-177.338,7.126,148.556
C05045=1182.500,243.506,-63.838,-177.340,7.124,148.557
C05046=1182.505,243.258,-63.811,-177.343,7.121,148.557
C05047=1182.509,243.009,-63.786,-177.345,7.119,148.557
C05048=1182.514,242.760,-63.759,-177.349,7.117,148.557
C05049=1182.518,242.512,-63.732,-177.351,7.115,148.557
C05050=1182.522,242.263,-63.706,-177.354,7.112,148.557
C05051=1182.526,242.015,-63.679,-177.356,7.110,148.558
C05052=1182.531,241.766,-63.653,-177.359,7.107,148.558
C05053=1182.535,241.517,-63.626,-177.362,7.105,148.558
C05054=1182.540,241.268,-63.600,-177.364,7.102,148.558
C05055=1182.544,241.020,-63.574,-177.367,7.100,148.558
C05056=1182.549,240.772,-63.548,-177.370,7.097,148.558
C05057=1182.554,240.524,-63.521,-177.372,7.095,148.558
C05058=1182.558,240.275,-63.495,-177.375,7.092,148.559
C05059=1182.563,240.026,-63.468,-177.377,7.090,148.559
C05060=1182.567,239.777,-63.443,-177.380,7.088,148.559
C05061=1182.571,239.529,-63.416,-177.383,7.085,148.559
C05062=1182.576,239.280,-63.390,-177.386,7.083,148.560
C05063=1182.580,239.031,-63.364,-177.388,7.081,148.560
C05064=1182.585,238.783,-63.337,-177.391,7.078,148.560
C05065=1182.589,238.535,-63.312,-177.393,7.076,148.560
C05066=1182.593,238.287,-63.285,-177.396,7.074,148.560
C05067=1182.598,238.037,-63.259,-177.399,7.071,148.560
C05068=1182.602,237.789,-63.233,-177.401,7.069,148.560
C05069=1182.606,237.540,-63.207,-177.404,7.066,148.561
C05070=1182.611,237.291,-63.180,-177.406,7.064,148.561
C05071=1182.616,237.043,-63.155,-177.409,7.061,148.561
C05072=1182.621,236.772,-63.126,-177.412,7.059,148.561
C05073=1182.626,236.500,-63.097,-177.415,7.057,148.562
C05074=1182.630,236.228,-63.069,-177.418,7.054,148.562
C05075=1182.635,235.957,-63.041,-177.421,7.051,148.562
C05076=1182.641,235.708,-63.015,-177.423,7.049,148.562
C05077=1182.645,235.460,-62.988,-177.426,7.046,148.562
C05078=1182.649,235.211,-62.962,-177.428,7.044,148.562
C05079=1182.653,234.962,-62.937,-177.431,7.042,148.563
C05080=1182.658,234.713,-62.910,-177.434,7.039,148.563
C05081=1182.662,234.466,-62.884,-177.436,7.038,148.563
C05082=1182.667,234.217,-62.858,-177.439,7.035,148.563
C05083=1182.671,233.968,-62.833,-177.442,7.033,148.564
C05084=1182.675,233.719,-62.807,-177.445,7.030,148.564
C05085=1182.680,233.470,-62.781,-177.447,7.028,148.564
C05086=1182.685,233.222,-62.755,-177.449,7.026,148.564
C05087=1182.689,232.973,-62.730,-177.453,7.023,148.564
C05088=1182.693,232.725,-62.704,-177.455,7.021,148.564
C05089=1182.697,232.476,-62.677,-177.458,7.018,148.565
C05090=1182.703,232.228,-62.651,-177.460,7.016,148.565
C05091=1182.707,231.979,-62.626,-177.463,7.014,148.565
C05092=1182.711,231.730,-62.600,-177.466,7.011,148.565
C05093=1182.716,231.482,-62.574,-177.468,7.010,148.566
C05094=1182.720,231.233,-62.549,-177.471,7.007,148.566
C05095=1182.725,230.985,-62.523,-177.474,7.005,148.566
C05096=1182.729,230.736,-62.497,-177.476,7.002,148.566
C05097=1182.734,230.487,-62.471,-177.479,7.000,148.566
C05098=1182.739,230.239,-62.445,-177.481,6.998,148.566
C05099=1182.743,229.990,-62.420,-177.484,6.995,148.567
C05100=1182.748,229.742,-62.394,-177.487,6.993,148.567
C05101=1182.752,229.493,-62.369,-177.490,6.991,148.567
C05102=1182.756,229.244,-62.343,-177.492,6.988,148.567
C05103=1182.761,228.996,-62.317,-177.495,6.987,148.568
C05104=1182.765,228.747,-62.292,-177.497,6.984,148.568
C05105=1182.770,228.498,-62.267,-177.500,6.982,148.568
C05106=1182.774,228.250,-62.241,-177.503,6.979,148.568
C05107=1182.779,228.001,-62.215,-177.505,6.977,148.568
C05108=1182.783,227.752,-62.190,-177.508,6.975,148.569
C05109=1182.788,227.504,-62.164,-177.511,6.972,148.569
C05110=1182.792,227.255,-62.139,-177.513,6.970,148.569
C05111=1182.796,227.006,-62.113,-177.516,6.968,148.569
C05112=1182.801,226.758,-62.088,-177.519,6.966,148.570
C05113=1182.806,226.509,-62.062,-177.521,6.964,148.570
C05114=1182.810,226.260,-62.037,-177.524,6.961,148.570
C05115=1182.815,226.012,-62.011,-177.526,6.959,148.570
C05116=1182.819,225.763,-61.986,-177.529,6.957,148.570
C05117=1182.824,225.514,-61.961,-177.532,6.954,148.570
C05118=1182.828,225.266,-61.935,-177.535,6.952,148.571
C05119=1182.832,225.017,-61.909,-177.537,6.950,148.571
C05120=1182.838,224.768,-61.885,-177.540,6.947,148.571
C05121=1182.842,224.519,-61.859,-177.543,6.946,148.572
C05122=1182.847,224.271,-61.834,-177.545,6.943,148.572
C05123=1182.851,224.022,-61.808,-177.548,6.941,148.572
C05124=1182.855,223.773,-61.783,-177.551,6.939,148.572
C05125=1182.859,223.525,-61.758,-177.553,6.936,148.572
C05126=1182.864,223.276,-61.732,-177.556,6.934,148.573
C05127=1182.869,223.028,-61.708,-177.558,6.932,148.573
C05128=1182.873,222.779,-61.682,-177.561,6.929,148.573
C05129=1182.878,222.530,-61.657,-177.564,6.927,148.573
C05130=1182.882,222.281,-61.631,-177.566,6.925,148.574
C05131=1182.887,222.033,-61.606,-177.569,6.923,148.574
C05132=1182.891,221.784,-61.582,-177.572,6.921,148.574
C05133=1182.895,221.535,-61.556,-177.574,6.919,148.574
C05134=1182.900,221.286,-61.531,-177.577,6.916,148.574
C05135=1182.905,221.038,-61.505,-177.580,6.914,148.575
C05136=1182.910,220.789,-61.481,-177.582,6.912,148.575
C05137=1182.913,220.540,-61.456,-177.585,6.909,148.575
C05138=1182.918,220.292,-61.431,-177.588,6.908,148.575
C05139=1182.923,220.043,-61.405,-177.590,6.906,148.576
C05140=1182.928,219.794,-61.380,-177.593,6.903,148.576
C05141=1182.931,219.546,-61.355,-177.596,6.901,148.576
C05142=1182.936,219.297,-61.331,-177.598,6.899,148.576
C05143=1182.941,219.048,-61.305,-177.601,6.896,148.577
C05144=1182.946,218.799,-61.280,-177.604,6.894,148.577
C05145=1182.949,218.551,-61.255,-177.606,6.892,148.577
C05146=1182.954,218.302,-61.230,-177.609,6.890,148.577
C05147=1182.959,218.054,-61.206,-177.612,6.888,148.578
C05148=1182.964,217.805,-61.180,-177.614,6.886,148.578
C05149=1182.968,217.556,-61.156,-177.617,6.883,148.578
C05150=1182.972,217.307,-61.130,-177.620,6.881,148.578
C05151=1182.977,217.059,-61.106,-177.622,6.879,148.579
C05152=1182.981,216.810,-61.081,-177.625,6.876,148.579
C05153=1182.986,216.562,-61.056,-177.628,6.874,148.579
C05154=1182.991,216.312,-61.031,-177.630,6.873,148.579
C05155=1182.995,216.064,-61.007,-177.633,6.871,148.580
C05156=1183.000,215.815,-60.982,-177.636,6.868,148.580
C05157=1183.004,215.566,-60.957,-177.638,6.866,148.580
C05158=1183.009,215.318,-60.932,-177.641,6.864,148.580
C05159=1183.013,215.068,-60.907,-177.644,6.861,148.580
C05160=1183.017,214.821,-60.882,-177.646,6.859,148.581
C05161=1183.022,214.572,-60.858,-177.649,6.858,148.581
C05162=1183.027,214.322,-60.833,-177.652,6.855,148.581
C05163=1183.031,214.074,-60.808,-177.654,6.853,148.582
C05164=1183.036,213.825,-60.783,-177.657,6.851,148.582
C05165=1183.040,213.577,-60.759,-177.659,6.849,148.582
C05166=1183.045,213.328,-60.734,-177.662,6.846,148.582
C05167=1183.049,213.079,-60.710,-177.665,6.844,148.583
C05168=1183.054,212.830,-60.685,-177.667,6.842,148.583
C05169=1183.059,212.581,-60.660,-177.671,6.840,148.583
C05170=1183.063,212.332,-60.636,-177.673,6.838,148.583
C05171=1183.068,212.084,-60.611,-177.675,6.836,148.584
C05172=1183.072,211.836,-60.586,-177.678,6.834,148.584
C05173=1183.077,211.586,-60.561,-177.681,6.831,148.584
C05174=1183.081,211.338,-60.537,-177.684,6.829,148.585
C05175=1183.086,211.089,-60.513,-177.686,6.827,148.585
C05176=1183.090,210.819,-60.486,-177.689,6.825,148.585
C05177=1183.095,210.549,-60.459,-177.692,6.823,148.585
C05178=1183.101,210.278,-60.433,-177.695,6.820,148.586
C05179=1183.105,210.007,-60.406,-177.698,6.819,148.586
C05180=1183.110,209.758,-60.382,-177.701,6.816,148.586
C05181=1183.115,209.510,-60.358,-177.703,6.814,148.586
C05182=1183.119,209.261,-60.333,-177.706,6.812,148.587
C05183=1183.124,209.012,-60.308,-177.709,6.809,148.587
C05184=1183.128,208.764,-60.284,-177.711,6.807,148.587
C05185=1183.133,208.515,-60.260,-177.714,6.805,148.588
C05186=1183.137,208.266,-60.235,-177.717,6.804,148.588
C05187=1183.142,208.017,-60.211,-177.719,6.801,148.588
C05188=1183.147,207.769,-60.186,-177.722,6.799,148.588
C05189=1183.151,207.520,-60.162,-177.725,6.797,148.589
C05190=1183.155,207.271,-60.137,-177.727,6.795,148.589
C05191=1183.160,207.022,-60.114,-177.730,6.792,148.589
C05192=1183.165,206.773,-60.090,-177.733,6.790,148.589
C05193=1183.170,206.525,-60.065,-177.735,6.789,148.590
C05194=1183.173,206.275,-60.041,-177.738,6.787,148.590
C05195=1183.179,206.027,-60.016,-177.741,6.784,148.590
C05196=1183.183,205.778,-59.992,-177.744,6.782,148.591
C05197=1183.188,205.529,-59.969,-177.746,6.780,148.591
C05198=1183.193,205.281,-59.944,-177.748,6.778,148.591
C05199=1183.197,205.031,-59.920,-177.751,6.776,148.591
C05200=1183.201,204.783,-59.896,-177.754,6.774,148.592
C05201=1183.205,204.535,-59.871,-177.756,6.772,148.592
C05202=1183.211,204.285,-59.848,-177.759,6.770,148.592
C05203=1183.215,204.037,-59.823,-177.762,6.768,148.592
C05204=1183.219,203.788,-59.799,-177.765,6.765,148.593
C05205=1183.224,203.539,-59.776,-177.767,6.763,148.593
C05206=1183.229,203.290,-59.751,-177.770,6.761,148.593
C05207=1183.233,203.042,-59.727,-177.773,6.760,148.594
C05208=1183.238,202.793,-59.703,-177.775,6.758,148.594
C05209=1183.242,202.544,-59.679,-177.778,6.755,148.594
C05210=1183.247,202.295,-59.654,-177.781,6.753,148.594
C05211=1183.251,202.046,-59.630,-177.783,6.751,148.595
C05212=1183.256,201.797,-59.607,-177.786,6.750,148.595
C05213=1183.260,201.549,-59.583,-177.789,6.747,148.595
C05214=1183.265,201.300,-59.560,-177.791,6.745,148.596
C05215=1183.270,201.051,-59.535,-177.794,6.743,148.596
C05216=1183.275,200.803,-59.511,-177.797,6.741,148.596
C05217=1183.279,200.553,-59.487,-177.799,6.739,148.597
C05218=1183.283,200.305,-59.463,-177.802,6.736,148.597
C05219=1183.288,200.055,-59.440,-177.805,6.735,148.597
C05220=1183.292,199.807,-59.416,-177.807,6.733,148.597
C05221=1183.297,199.558,-59.392,-177.810,6.731,148.598
C05222=1183.302,199.309,-59.368,-177.812,6.729,148.598
C05223=1183.307,199.060,-59.344,-177.816,6.726,148.598
C05224=1183.311,198.812,-59.320,-177.818,6.724,148.598
C05225=1183.316,198.563,-59.297,-177.821,6.723,148.599
C05226=1183.320,198.314,-59.273,-177.824,6.721,148.599
C05227=1183.324,198.065,-59.249,-177.826,6.719,148.599
C05228=1183.329,197.816,-59.225,-177.828,6.717,148.600
C05229=1183.333,197.567,-59.202,-177.832,6.714,148.600
C05230=1183.338,197.319,-59.177,-177.834,6.713,148.600
C05231=1183.342,197.070,-59.154,-177.837,6.711,148.601
C05232=1183.347,196.821,-59.131,-177.839,6.709,148.601
C05233=1183.352,196.572,-59.106,-177.842,6.707,148.601
C05234=1183.357,196.323,-59.083,-177.844,6.705,148.601
C05235=1183.361,196.075,-59.059,-177.848,6.702,148.602
C05236=1183.366,195.826,-59.035,-177.850,6.701,148.602
C05237=1183.371,195.577,-59.012,-177.853,6.699,148.602
C05238=1183.375,195.328,-58.988,-177.855,6.697,148.603
C05239=1183.380,195.079,-58.964,-177.858,6.695,148.603
C05240=1183.385,194.830,-58.941,-177.861,6.693,148.603
C05241=1183.389,194.581,-58.918,-177.864,6.691,148.604
C05242=1183.394,194.333,-58.894,-177.866,6.688,148.604
C05243=1183.398,194.084,-58.870,-177.869,6.687,148.604
C05244=1183.402,193.835,-58.848,-177.871,6.685,148.604
C05245=1183.407,193.586,-58.823,-177.874,6.683,148.605
C05246=1183.411,193.337,-58.800,-177.877,6.681,148.605
C05247=1183.416,193.088,-58.777,-177.880,6.679,148.606
C05248=1183.421,192.839,-58.753,-177.882,6.676,148.606
C05249=1183.426,192.590,-58.730,-177.885,6.675,148.606
C05250=1183.430,192.342,-58.706,-177.887,6.673,148.606
C05251=1183.435,192.093,-58.683,-177.890,6.671,148.607
C05252=1183.439,191.844,-58.659,-177.893,6.669,148.607
C05253=1183.444,191.595,-58.636,-177.895,6.668,148.607
C05254=1183.449,191.346,-58.613,-177.898,6.665,148.608
C05255=1183.453,191.097,-58.589,-177.901,6.663,148.608
C05256=1183.457,190.849,-58.566,-177.903,6.661,148.608
C05257=1183.462,190.600,-58.543,-177.906,6.659,148.609
C05258=1183.467,190.351,-58.519,-177.909,6.657,148.609
C05259=1183.472,190.102,-58.496,-177.911,6.656,148.609
C05260=1183.477,189.853,-58.473,-177.914,6.654,148.610
C05261=1183.481,189.604,-58.449,-177.916,6.652,148.610
C05262=1183.486,189.355,-58.426,-177.920,6.649,148.610
C05263=1183.490,189.106,-58.403,-177.922,6.647,148.610
C05264=1183.495,188.857,-58.380,-177.925,6.646,148.611
C05265=1183.499,188.608,-58.356,-177.928,6.644,148.611
C05266=1183.504,188.359,-58.333,-177.930,6.642,148.611
C05267=1183.509,188.111,-58.310,-177.933,6.640,148.612
C05268=1183.513,187.862,-58.287,-177.935,6.638,148.612
C05269=1183.518,187.613,-58.264,-177.938,6.636,148.612
C05270=1183.523,187.364,-58.241,-177.941,6.634,148.613
C05271=1183.527,187.115,-58.217,-177.944,6.632,148.613
C05272=1183.531,186.866,-58.194,-177.946,6.630,148.613
C05273=1183.536,186.617,-58.171,-177.949,6.628,148.614
C05274=1183.541,186.368,-58.148,-177.952,6.626,148.614
C05275=1183.546,186.120,-58.125,-177.954,6.624,148.614
C05276=1183.550,185.871,-58.102,-177.957,6.623,148.615
C05277=1183.555,185.622,-58.079,-177.959,6.621,148.615
C05278=1183.560,185.373,-58.056,-177.962,6.619,148.615
C05279=1183.564,185.124,-58.033,-177.965,6.617,148.616
C05280=1183.569,184.854,-58.008,-177.968,6.615,148.616
C05281=1183.574,184.585,-57.982,-177.970,6.613,148.616
C05282=1183.579,184.316,-57.958,-177.973,6.611,148.617
C05283=1183.584,184.046,-57.933,-177.976,6.608,148.617
C05284=1183.588,183.797,-57.910,-177.979,6.607,148.617
C05285=1183.593,183.548,-57.888,-177.982,6.605,148.618
C05286=1183.598,183.299,-57.865,-177.984,6.603,148.618
C05287=1183.602,183.050,-57.842,-177.987,6.601,148.618
C05288=1183.607,182.801,-57.818,-177.990,6.599,148.619
C05289=1183.612,182.552,-57.796,-177.992,6.598,148.619
C05290=1183.616,182.304,-57.773,-177.995,6.596,148.619
C05291=1183.621,182.055,-57.750,-177.997,6.594,148.620
C05292=1183.625,181.806,-57.727,-178.000,6.592,148.620
C05293=1183.630,181.556,-57.705,-178.003,6.589,148.620
C05294=1183.635,181.308,-57.682,-178.006,6.588,148.621
C05295=1183.639,181.059,-57.659,-178.009,6.586,148.621
C05296=1183.644,180.810,-57.636,-178.011,6.584,148.621
C05297=1183.648,180.561,-57.613,-178.014,6.582,148.622
C05298=1183.654,180.313,-57.590,-178.017,6.580,148.622
C05299=1183.658,180.063,-57.568,-178.019,6.579,148.622
C05300=1183.663,179.814,-57.545,-178.022,6.577,148.623
C05301=1183.667,179.566,-57.523,-178.025,6.575,148.623
C05302=1183.672,179.316,-57.500,-178.027,6.573,148.623
C05303=1183.676,179.068,-57.477,-178.029,6.571,148.624
C05304=1183.681,178.818,-57.455,-178.032,6.569,148.624
C05305=1183.686,178.570,-57.432,-178.035,6.568,148.624
C05306=1183.690,178.321,-57.409,-178.037,6.566,148.625
C05307=1183.695,178.072,-57.387,-178.040,6.564,148.625
C05308=1183.700,177.823,-57.364,-178.043,6.562,148.626
C05309=1183.704,177.574,-57.342,-178.046,6.561,148.626
C05310=1183.709,177.325,-57.318,-178.048,6.559,148.626
C05311=1183.714,177.076,-57.297,-178.051,6.556,148.627
C05312=1183.718,176.827,-57.273,-178.054,6.554,148.627
C05313=1183.723,176.578,-57.251,-178.057,6.553,148.627
C05314=1183.727,176.330,-57.229,-178.059,6.551,148.628
C05315=1183.732,176.080,-57.206,-178.062,6.549,148.628
C05316=1183.737,175.831,-57.184,-178.065,6.547,148.628
C05317=1183.742,175.583,-57.161,-178.067,6.545,148.629
C05318=1183.746,175.333,-57.139,-178.070,6.544,148.629
C05319=1183.750,175.085,-57.116,-178.073,6.542,148.629
C05320=1183.756,174.836,-57.094,-178.075,6.540,148.630
C05321=1183.760,174.587,-57.071,-178.078,6.538,148.630
C05322=1183.765,174.338,-57.049,-178.080,6.536,148.630
C05323=1183.770,174.089,-57.027,-178.083,6.534,148.631
C05324=1183.773,173.840,-57.004,-178.086,6.533,148.631
C05325=1183.779,173.591,-56.982,-178.088,6.531,148.631
C05326=1183.783,173.342,-56.960,-178.091,6.529,148.632
C05327=1183.788,173.094,-56.938,-178.094,6.527,148.632
C05328=1183.793,172.844,-56.915,-178.096,6.526,148.633
C05329=1183.797,172.595,-56.893,-178.099,6.524,148.633
C05330=1183.802,172.347,-56.870,-178.102,6.522,148.633
C05331=1183.807,172.097,-56.848,-178.104,6.520,148.634
C05332=1183.812,171.848,-56.826,-178.107,6.518,148.634
C05333=1183.816,171.599,-56.804,-178.110,6.517,148.634
C05334=1183.820,171.350,-56.781,-178.112,6.515,148.635
C05335=1183.825,171.101,-56.759,-178.115,6.513,148.635
C05336=1183.830,170.852,-56.737,-178.118,6.511,148.635
C05337=1183.835,170.603,-56.715,-178.121,6.510,148.636
C05338=1183.839,170.355,-56.693,-178.123,6.508,148.636
C05339=1183.844,170.106,-56.670,-178.126,6.506,148.637
C05340=1183.848,169.856,-56.648,-178.129,6.504,148.637
C05341=1183.853,169.608,-56.627,-178.131,6.502,148.637
C05342=1183.858,169.358,-56.605,-178.134,6.501,148.638
C05343=1183.863,169.109,-56.582,-178.137,6.499,148.638
C05344=1183.867,168.861,-56.559,-178.139,6.497,148.638
C05345=1183.872,168.612,-56.538,-178.142,6.495,148.639
C05346=1183.876,168.363,-56.516,-178.145,6.494,148.639
C05347=1183.881,168.114,-56.494,-178.147,6.492,148.639
C05348=1183.886,167.864,-56.471,-178.150,6.490,148.640
C05349=1183.891,167.616,-56.450,-178.153,6.488,148.640
C05350=1183.895,167.366,-56.428,-178.155,6.486,148.641
C05351=1183.900,167.118,-56.406,-178.158,6.485,148.641
C05352=1183.904,166.868,-56.384,-178.161,6.483,148.641
C05353=1183.909,166.620,-56.362,-178.163,6.481,148.642
C05354=1183.914,166.370,-56.340,-178.166,6.479,148.642
C05355=1183.919,166.121,-56.318,-178.168,6.478,148.642
C05356=1183.923,165.872,-56.296,-178.171,6.477,148.643
C05357=1183.928,165.623,-56.274,-178.174,6.475,148.643
C05358=1183.933,165.374,-56.252,-178.176,6.473,148.644
C05359=1183.937,165.125,-56.231,-178.179,6.471,148.644
C05360=1183.942,164.877,-56.209,-178.182,6.469,148.644
C05361=1183.947,164.627,-56.187,-178.184,6.468,148.645
C05362=1183.951,164.379,-56.165,-178.187,6.466,148.645
C05363=1183.956,164.130,-56.143,-178.190,6.464,148.645
C05364=1183.961,163.881,-56.121,-178.192,6.462,148.646
C05365=1183.965,163.632,-56.099,-178.195,6.461,148.646
C05366=1183.970,163.383,-56.078,-178.198,6.459,148.646
C05367=1183.975,163.134,-56.056,-178.200,6.457,148.647
C05368=1183.979,162.885,-56.034,-178.203,6.456,148.647
C05369=1183.984,162.636,-56.013,-178.206,6.454,148.648
C05370=1183.988,162.386,-55.991,-178.209,6.452,148.648
C05371=1183.993,162.138,-55.969,-178.212,6.450,148.649
C05372=1183.998,161.889,-55.948,-178.214,6.449,148.649
C05373=1184.002,161.640,-55.925,-178.216,6.448,148.649
C05374=1184.007,161.391,-55.904,-178.219,6.446,148.650
C05375=1184.012,161.141,-55.882,-178.222,6.444,148.650
C05376=1184.017,160.892,-55.861,-178.224,6.442,148.650
C05377=1184.021,160.644,-55.839,-178.227,6.441,148.651
C05378=1184.026,160.394,-55.817,-178.230,6.439,148.651
C05379=1184.031,160.145,-55.796,-178.232,6.437,148.652
C05380=1184.036,159.897,-55.774,-178.235,6.435,148.652
C05381=1184.040,159.647,-55.752,-178.238,6.433,148.652
C05382=1184.045,159.399,-55.731,-178.240,6.432,148.653
C05383=1184.050,159.149,-55.710,-178.243,6.430,148.653
C05384=1184.055,158.881,-55.686,-178.246,6.428,148.654
C05385=1184.060,158.612,-55.663,-178.249,6.427,148.654
C05386=1184.065,158.342,-55.640,-178.252,6.425,148.654
C05387=1184.070,158.074,-55.616,-178.254,6.423,148.655
C05388=1184.075,157.824,-55.595,-178.257,6.421,148.655
C05389=1184.079,157.575,-55.573,-178.260,6.420,148.656
C05390=1184.084,157.326,-55.553,-178.263,6.418,148.656
C05391=1184.089,157.078,-55.531,-178.266,6.416,148.656
C05392=1184.093,156.828,-55.509,-178.268,6.415,148.657
C05393=1184.098,156.579,-55.488,-178.271,6.413,148.657
C05394=1184.103,156.330,-55.466,-178.274,6.411,148.658
C05395=1184.108,156.081,-55.445,-178.276,6.410,148.658
C05396=1184.112,155.832,-55.424,-178.278,6.408,148.658
C05397=1184.117,155.583,-55.402,-178.281,6.407,148.659
C05398=1184.122,155.334,-55.381,-178.284,6.405,148.659
C05399=1184.127,155.085,-55.360,-178.286,6.403,148.660
C05400=1184.131,154.836,-55.338,-178.289,6.401,148.660
C05401=1184.135,154.587,-55.317,-178.292,6.400,148.660
C05402=1184.141,154.338,-55.296,-178.295,6.398,148.661
C05403=1184.145,154.089,-55.274,-178.298,6.396,148.661
C05404=1184.150,153.839,-55.253,-178.300,6.395,148.662
C05405=1184.155,153.591,-55.231,-178.303,6.394,148.662
C05406=1184.159,153.342,-55.211,-178.305,6.392,148.662
C05407=1184.164,153.093,-55.189,-178.308,6.390,148.663
C05408=1184.169,152.843,-55.168,-178.311,6.388,148.663
C05409=1184.174,152.594,-55.147,-178.313,6.387,148.664
C05410=1184.178,152.346,-55.126,-178.316,6.385,148.664
C05411=1184.183,152.096,-55.105,-178.319,6.383,148.664
C05412=1184.188,151.848,-55.083,-178.321,6.382,148.665
C05413=1184.192,151.598,-55.063,-178.324,6.381,148.665
C05414=1184.197,151.349,-55.042,-178.327,6.379,148.666
C05415=1184.202,151.100,-55.020,-178.329,6.377,148.666
C05416=1184.206,150.851,-55.000,-178.332,6.375,148.666
C05417=1184.212,150.602,-54.979,-178.335,6.374,148.667
C05418=1184.216,150.353,-54.957,-178.337,6.372,148.667
C05419=1184.220,150.104,-54.936,-178.340,6.371,148.668
C05420=1184.225,149.854,-54.915,-178.343,6.370,148.668
C05421=1184.230,149.606,-54.894,-178.345,6.368,148.669
C05422=1184.235,149.357,-54.873,-178.348,6.366,148.669
C05423=1184.240,149.108,-54.852,-178.351,6.364,148.669
C05424=1184.245,148.859,-54.831,-178.353,6.362,148.670
C05425=1184.249,148.609,-54.810,-178.355,6.361,148.670
C05426=1184.254,148.360,-54.789,-178.358,6.360,148.670
C05427=1184.258,148.111,-54.768,-178.361,6.358,148.671
C05428=1184.263,147.862,-54.747,-178.364,6.357,148.671
C05429=1184.268,147.613,-54.726,-178.367,6.355,148.672
C05430=1184.273,147.364,-54.705,-178.369,6.353,148.672
C05431=1184.278,147.115,-54.684,-178.372,6.351,148.673
C05432=1184.282,146.866,-54.664,-178.374,6.350,148.673
C05433=1184.287,146.617,-54.643,-178.377,6.349,148.673
C05434=1184.291,146.368,-54.622,-178.380,6.347,148.674
C05435=1184.296,146.118,-54.601,-178.383,6.345,148.674
C05436=1184.301,145.869,-54.580,-178.385,6.344,148.675
C05437=1184.306,145.620,-54.559,-178.388,6.343,148.675
C05438=1184.310,145.371,-54.539,-178.390,6.341,148.675
C05439=1184.315,145.122,-54.518,-178.393,6.339,148.676
C05440=1184.320,144.873,-54.498,-178.396,6.338,148.676
C05441=1184.325,144.624,-54.477,-178.399,6.336,148.677
C05442=1184.329,144.375,-54.456,-178.401,6.334,148.677
C05443=1184.334,144.126,-54.435,-178.404,6.333,148.678
C05444=1184.339,143.877,-54.414,-178.406,6.332,148.678
C05445=1184.344,143.628,-54.393,-178.409,6.330,148.678
C05446=1184.348,143.379,-54.373,-178.412,6.328,148.679
C05447=1184.354,143.130,-54.352,-178.415,6.327,148.679
C05448=1184.358,142.881,-54.332,-178.417,6.326,148.680
C05449=1184.362,142.631,-54.311,-178.420,6.324,148.680
C05450=1184.367,142.382,-54.290,-178.422,6.322,148.681
C05451=1184.371,142.133,-54.269,-178.425,6.320,148.681
C05452=1184.377,141.884,-54.249,-178.428,6.319,148.682
C05453=1184.381,141.635,-54.228,-178.430,6.318,148.682
C05454=1184.386,141.385,-54.207,-178.433,6.316,148.682
C05455=1184.391,141.137,-54.187,-178.436,6.314,148.683
C05456=1184.395,140.888,-54.166,-178.438,6.313,148.683
C05457=1184.401,140.638,-54.146,-178.442,6.311,148.684
C05458=1184.405,140.389,-54.126,-178.444,6.310,148.684
C05459=1184.409,140.140,-54.105,-178.446,6.309,148.685
C05460=1184.415,139.891,-54.084,-178.449,6.307,148.685
C05461=1184.419,139.642,-54.064,-178.452,6.305,148.685
C05462=1184.424,139.393,-54.044,-178.454,6.304,148.686
C05463=1184.429,139.144,-54.023,-178.457,6.303,148.686
C05464=1184.434,138.895,-54.003,-178.460,6.301,148.687
C05465=1184.438,138.646,-53.983,-178.462,6.299,148.687
C05466=1184.444,138.396,-53.962,-178.465,6.297,148.687
C05467=1184.448,138.147,-53.942,-178.467,6.297,148.688
C05468=1184.453,137.898,-53.921,-178.470,6.295,148.688
C05469=1184.458,137.649,-53.900,-178.473,6.293,148.689
C05470=1184.462,137.400,-53.880,-178.476,6.292,148.689
C05471=1184.467,137.151,-53.860,-178.478,6.291,148.690
C05472=1184.471,136.902,-53.840,-178.481,6.289,148.690
C05473=1184.476,136.652,-53.819,-178.484,6.288,148.691
C05474=1184.481,136.403,-53.799,-178.487,6.286,148.691
C05475=1184.486,136.154,-53.779,-178.489,6.285,148.691
